# B&R Automation Studio project NAELD004C00R10L518F00 (part 47)

#### Act_InitLocal.st
```iecst
(** 2019-04-16 **)
ACTION Act_InitLocal:

	//Input Reference Link To Local Variable
	p_udiRstErr ACCESS ADR(udiRstErr);
	p_bEn ACCESS ADR(bEn);
	p_bDis ACCESS ADR(bDis);
	p_bRun ACCESS ADR(bRun);
	p_bStop ACCESS ADR(bStop);
	p_bStep ACCESS ADR(bStep);

	p_sProgNm ACCESS ADR(sProgNm);
	p_bNtSettingsLoadDone ACCESS ADR(bNtSettingsLoadDone);

	p_usiMagConv ACCESS ADR(usiMagConv);
	p_bInfoEn ACCESS ADR(bInfoEn);
	p_bInfoMag1Mty ACCESS ADR(bInfoMag1Mty);
	p_bInfoMag2Mty ACCESS ADR(bInfoMag2Mty);
	p_bInfoMag3Mty ACCESS ADR(bInfoMag3Mty);

	pa_bMagDis ACCESS ADR(a_bMagDis);

	p_bNewMag ACCESS ADR(bNewMag);
	p_bRlsMag ACCESS ADR(bRlsMag);

	p_bUSAllow ACCESS ADR(bUSAllow);
	p_tyBufferStat1 ACCESS ADR(tyBufferStat1);
	p_tyBufferStat2 ACCESS ADR(tyBufferStat2);
	p_tyBufferStat3 ACCESS ADR(tyBufferStat3);
	p_tyBufferStat4 ACCESS ADR(tyBufferStat4);

	p_bMagClampRS1 ACCESS ADR(bMagClampRS1);
	p_bMagClampRS2 ACCESS ADR(bMagClampRS2);
	p_bMagClampRS3 ACCESS ADR(bMagClampRS3);
	p_bMagClampRS4 ACCESS ADR(bMagClampRS4);

	p_bMagEntrySen1 ACCESS ADR(bMagEntrySen1);
	p_bMagEntrySen2 ACCESS ADR(bMagEntrySen2);
	p_bMagEntrySen3 ACCESS ADR(bMagEntrySen3);
	p_bMagEntrySen4 ACCESS ADR(bMagEntrySen4);

	p_bMagPresentSen1 ACCESS ADR(bMagPresentSen1);
	p_bMagPresentSen2 ACCESS ADR(bMagPresentSen2);
	p_bMagPresentSen3 ACCESS ADR(bMagPresentSen3);
	p_bMagPresentSen4 ACCESS ADR(bMagPresentSen4);

	p_bBufferMagPresent1 ACCESS ADR(bBufferMagPresent1);
	p_bBufferMagPresent2 ACCESS ADR(bBufferMagPresent2);
	p_bBufferMagPresent3 ACCESS ADR(bBufferMagPresent3);
	p_bBufferMagPresent4 ACCESS ADR(bBufferMagPresent4);

	p_dtBufferMagPresentTm1 ACCESS ADR(dtBufferMagPresentTm1);
	p_dtBufferMagPresentTm2 ACCESS ADR(dtBufferMagPresentTm2);
	p_dtBufferMagPresentTm3 ACCESS ADR(dtBufferMagPresentTm3);
	p_dtBufferMagPresentTm4 ACCESS ADR(dtBufferMagPresentTm4);

	p_eBufferStat ACCESS ADR(eBufferStat);
	p_eBufferStatus ACCESS ADR(eBufferStatus);

	p_eMagConv2ClpStat ACCESS ADR(eMagConv2ClpStat);
	p_eMagConv2ClpStatus ACCESS ADR(eMagConv2ClpStatus);
	p_bMagConv2ClpHvMag ACCESS ADR(bMagConv2ClpHvMag);

	p_eDSSMEMAStat ACCESS ADR(eDSSMEMAStat);
	p_eDSSMEMAStatus ACCESS ADR(eDSSMEMAStatus);
	p_bDSSMEMAConvStart ACCESS ADR(bDSSMEMAConvStart);

	p_eAGVMagStat ACCESS ADR(eAGVMagStat);
	p_eAGVMagStatus ACCESS ADR(eAGVMagStatus);
	p_bAGVMagMcRunRdy ACCESS ADR(bAGVMagMcRunRdy);
	p_tyAGVToDTMag ACCESS ADR(tyAGVToDTMag);

	p_eTrolleyLckStat ACCESS ADR(eTrolleyLckStat);
	p_eTrolleyLckStatus ACCESS ADR(eTrolleyLckStatus);

END_ACTION
```

#### Act_Link.st
```iecst
(** 2018-12-11 **)
ACTION Act_Link:

	IF p_eLinkMag = LDMagQuadruple = FALSE THEN
		//Sensor
		p_bMagPresentSen1	:= p_bLinkDIMagPresentSen1 OR p_bLinkMagConv2Clp1MtrIn OR p_bLinkMagConv2Clp1MtrOut;
		p_bMagPresentSen2	:= p_bLinkDIMagPresentSen2 OR p_bLinkMagConv2Clp2MtrIn OR p_bLinkMagConv2Clp2MtrOut;
		p_bMagPresentSen3	:= p_bLinkDIMagPresentSen3 OR p_bLinkMagConv2Clp3MtrIn OR p_bLinkMagConv2Clp3MtrOut;
		p_bMagPresentSen4	:= p_bLinkDIMagPresentSen4 OR p_bLinkMagConv2Clp4MtrIn OR p_bLinkMagConv2Clp4MtrOut;

		//Clamp RS
		p_bMagClampRS1 		:= (p_bLinkFixedMagClampRS1 AND p_bLinkRmtMagClampRS1) OR p_bLinkNewMagVerified1;
		p_bMagClampRS2		:= (p_bLinkFixedMagClampRS2 AND p_bLinkRmtMagClampRS2) OR bNewMagVerified;
		p_bMagClampRS3		:= (p_bLinkFixedMagClampRS3 AND p_bLinkRmtMagClampRS3) OR p_bLinkNewMagVerified3;
		p_bMagClampRS4		:= (p_bLinkFixedMagClampRS4 AND p_bLinkRmtMagClampRS4) OR p_bLinkNewMagVerified4;

	ELSE
		IF p_eLinkMag = LDMagQuadruple THEN
			CASE p_usiLinkMod OF
				0,1:
					//Sensor
					p_bMagPresentSen1	:= p_bLinkDIMagPresentSen1 OR p_bLinkMagConv2Clp1MtrIn OR p_bLinkMagConv2Clp1MtrOut;
					p_bMagPresentSen2	:= p_bLinkDIMagPresentSen2 OR p_bLinkMagConv2Clp2MtrIn OR p_bLinkMagConv2Clp2MtrOut;
					p_bMagPresentSen3	:= p_bLinkDIMagPresentSen3 OR p_bLinkMagConv2Clp3MtrIn OR p_bLinkMagConv2Clp3MtrOut;
					p_bMagPresentSen4	:= p_bLinkDIMagPresentSen4 OR p_bLinkMagConv2Clp4MtrIn OR p_bLinkMagConv2Clp4MtrOut;

					//Clamp RS
					p_bMagClampRS1 		:= (p_bLinkFixedMagClampRS1 AND p_bLinkRmtMagClampRS1) OR p_bLinkNewMagVerified1;
					p_bMagClampRS2		:= (p_bLinkFixedMagClampRS2 AND p_bLinkRmtMagClampRS2) OR bNewMagVerified;
					p_bMagClampRS3		:= (p_bLinkFixedMagClampRS3 AND p_bLinkRmtMagClampRS3) OR p_bLinkNewMagVerified3;
					p_bMagClampRS4		:= (p_bLinkFixedMagClampRS4 AND p_bLinkRmtMagClampRS4) OR p_bLinkNewMagVerified4;

				2:
					//Sensor
					p_bMagPresentSen1	:= p_bLinkDIMagPresentSen1 OR p_bLinkMagConv2Clp1MtrIn OR p_bLinkMagConv2Clp1MtrOut;
					p_bMagPresentSen2	:= p_bLinkDIMagPresentSen2 OR p_bLinkMagConv2Clp2MtrIn OR p_bLinkMagConv2Clp2MtrOut;
					p_bMagPresentSen3	:= FALSE;
					p_bMagPresentSen4	:= FALSE;

					//Clamp RS
					p_bMagClampRS1 		:= (p_bLinkFixedMagClampRS1 AND p_bLinkRmtMagClampRS1) OR p_bLinkNewMagVerified1;
					p_bMagClampRS2		:= (p_bLinkFixedMagClampRS2 AND p_bLinkRmtMagClampRS2) OR bNewMagVerified;
					p_bMagClampRS3		:= FALSE;
					p_bMagClampRS4		:= FALSE;

			END_CASE
		END_IF
	END_IF

	//Mag Exchange Mode
	CASE p_eLinkMcParamMagExMode OF
		McSetMagXcAutoManMode:
			bMagManEx := TRUE;
			bMagAutoEx := TRUE;

		McSetMagXcAutoMode:
			bMagManEx := FALSE;
			bMagAutoEx := TRUE;

		McSetMagXcManMode:
			bMagManEx := TRUE;
			bMagAutoEx := FALSE;

	END_CASE

	//New magazine auto detection at inlet sensor
	fbMagAutoDetTm(IN := p_bLinkDIMagEntrySen OR p_bLinkDIMagPresentSen2, PT := DINT_TO_TIME(p_bLinkMcParamMagAutoDetTm));
	IF fbMagAutoDetTm.Q AND bMagManEx THEN
		bNewMagAutoDetected := TRUE;
	ELSE
		bNewMagAutoDetected := FALSE;
	END_IF

	//Front or rear lane magazine mode
	IF p_eLinkMag = LDMagQuadruple THEN
		CASE p_usiLinkMod OF
			0,2:
				usiMagModel := p_bLinkMagRcpCurrRcpMagModel;

			1:
				usiMagModel := p_bLinkMagRcpCurrRcpMagModel1;
		END_CASE

	ELSE
		usiMagModel := p_bLinkMagRcpCurrRcpMagModel;

	END_IF

	IF p_bLinkNtParamMagModelAutoVerify THEN
		IF usiMagModel = 0  //CAB706.2
			AND p_bDIMagConvHeightSen = TRUE
			AND p_bDIMagConvSelUnclampRS = FALSE
			AND p_bDIMagConvCAB717Sen = FALSE
			AND p_bDIMagConvSmallSen
			THEN
			bNewMagVerified:= TRUE;

		ELSIF  usiMagModel = 1 //CAB716.2
			AND p_bDIMagConvHeightSen = FALSE
			AND p_bDIMagConvSelUnclampRS = FALSE
			AND p_bDIMagConvCAB717Sen = FALSE
			AND p_bDIMagConvSmallSen
			THEN
			bNewMagVerified:= TRUE;

		ELSIF  usiMagModel = 2 //CAB717.2
			AND p_bDIMagConvHeightSen = FALSE
			AND p_bDIMagConvSelUnclampRS
			AND p_bDIMagConvCAB717Sen
			AND p_bDIMagConvLargeSen
			THEN
			bNewMagVerified:= TRUE;
		ELSE
			bNewMagVerified:= FALSE;
		END_IF
	ELSE
		bNewMagVerified:= TRUE;
	END_IF

	bAIVInPos := p_tyAGVToDTMag.bVEHInPos2 OR p_bDISOTRcv;

	IF p_bBufferMagRemoved THEN
		bManualUnloadMag := FALSE;
	END_IF

	IF EDGEPOS(p_bOpsTravLifULUpdatePullSlot) THEN
		bOpsTravLifULUpdatePullSlot := TRUE;
	ELSIF p_bOpsTravLifULUpdatePullSlot = FALSE THEN
		bOpsTravLifULUpdatePullSlot := FALSE;
	END_IF

	//Auto recipe
	IF p_bNtParamAutoRcpPrep THEN
		p_bUSAllow := NOT(p_bMagPropDiffBlk); //false
//		p_bAdaptFollowerBlk := p_sProdRcpCurrRcp1Name <>  p_sProdRcpCrZ2RcpNm;
	ELSE
		p_bUSAllow ACCESS p_Follower1USAllow;
//		p_bAdaptFollowerBlk := FALSE;
	END_IF

	//Trolley lock feature
	IF p_bLinkTrolleyLckPrep THEN
		fbTrllySenOff(IN:= p_bTrolleyPreSen=FALSE);
		IF EDGEPOS(p_bTrolleyPreSen) THEN
			eTrolleyLck :=  PneuActExt;
			bTrllyRetDone := FALSE;
		ELSIF eGotoOpsStep = MagConvLDStepMagUSComm AND eOpsStep = MagConvLDStepMagExitedWait OR p_bUITrolleyUnlck THEN
			eTrolleyLck :=  PneuActRet;
		ELSIF NOT(p_bTrolleyPreSen) AND fbTrllySenOff.Q AND bTrllyRetDone = FALSE THEN
			eTrolleyLck :=  PneuActRet;
			bTrllyRetDone := TRUE;
		END_IF
		IF p_eTrolleyLckStat = PneuActRet OR  p_eTrolleyLckStat = PneuActExt AND p_eTrolleyLckStatus = Done THEN
			eTrolleyLck :=  PneuActIdle;
			p_bUITrolleyUnlck := FALSE; //bi-dir
		END_IF
	END_IF
END_ACTION
```

#### Init.st
```iecst
(** 2019-03-25 **)
PROGRAM _INIT

	(* Always Change If Project Change *)

	//Physical Configuration
	usiMagConv	:= 2;

	//Pass Address To Global Address For External Use
	//Action, State & Status

	//Alarm
	p_OpsMagConvLD2AlmData	:= ADR(tyAlmData);
	p_OpsMagConvLD2AlmData1	:= ADR(tyAlmData1);

	//Output
	p_OpsMagConvLD2StepTxt	:= ADR(sStepTxt);
	p_OpsMagConvLD2Paused	:= ADR(bPaused);

	p_OpsMagConvLD2BufferAct		:= ADR(eBufferAct);
	p_OpsMagConvLD2MagConv2ClpAct	:= ADR(eMagConv2ClpAct);
	p_OpsMagConvLD2DSSMEMAAct		:= ADR(eDSSMEMAAct);
	p_OpsMagConvLD2AGVMagAct		:= ADR(eAGVMagAct);
	p_OpsMagConvLD2SafetyBarAct			:= ADR(eSafetyBarAct);

	p_OpsMagConvLD2InitDone				:= ADR(bOpsInitDone);
	p_OpsMagConvLD2MagBffrAvl			:= ADR(bMagBffrAvl);
	p_OpsMagConvLD2NewMagAllw			:= ADR(bNewMagAllw);
	p_OpsMagConvLD2RlsMagAllw			:= ADR(bRlsMagAllw);
	p_OpsMagConvLD2StepMagExitedWait	:= ADR(bStepMagExitedWait);
	p_OpsMagConvLD2StepUSCom			:= ADR(bStepMagUSCom);

	p_OpsMagConvLD2StepSelClampCtrl		:= ADR(eSelClampCtrl);

	p_OpsMagConvLD2NewMagVerified		:= ADR(bNewMagVerified);
	p_OpsMagConvLD2MagMtyExit			:= ADR(bStepMagMtyExit);
	p_OpsMagConvLD2IncorrectMagModel    := ADR(bIncorrectMagazineModel);
	p_OpsMagConvLD2MagSizeL    			:= ADR(bMagSizeLarge);

	p_OpsMagConvLD2USSOTAct			:= ADR(eUSSOTAct);
	p_OpsMagConvLD2DSSOTAct			:= ADR(eDSSOTAct);

	p_OpsMagConvLD2ExitedWait			:= ADR(bMagExitedWait);
	p_OpsMagConvLD2DSCom				:= ADR(bStepDSCom);
	p_OpsMagConvLD2AGVCommRdy			:= ADR(bAGVCommRdy);

	p_OpsMagConvLD2UnclmpDone			:= ADR(bPneuUnclmpDone);
	p_OpsMagConvLD2MagAllwGo			:= ADR(udiMagAllwGo);
	p_OpsMagConvLD2QueryWO 				:= ADR(bQueryWO);
	p_OpsMagConvLD2ReadRFID				:= ADR(bReadRFID);
	p_OpsMagConvLD2WriteRFID			:= ADR(bWriteRFID);
	p_OpsMagConvLD2ExtDelAutoRcp		:= ADR(bExitDelAutoRcp);
	p_OpsMagConvLD2RlsMagUmask			:= ADR(bRlsMagBtnUnmask);
	p_OpsMagConvLD2ExtMes				:= ADR(bExtMesStdByChk);
	p_OpsMagConvLD2HModChgDone			:= ADR(bHCommModChgDone);
	p_OpsMagConvLD2TrolleyLck			:= ADR(eTrolleyLck);

	(* Always Change If Project Change *)

END_PROGRAM
```

#### Program Logical/Operations/OpsMagConvLD2/Sequence

##### Act_LogStep.st
```iecst
(** 2019-03-25 **)
ACTION Act_LogStep:

//log
	IF EDGEPOS (bClsLog) THEN
		memset(ADR(logStep),0,SIZEOF(logStep));
		logIndexStep := 0;
		bClsLog := FALSE;
	END_IF

	blog := eOpsStep <> eGotoOpsStepDummy;

	IF blog THEN
		logStep[logIndexStep] := eOpsStep;
		logIndexStep := logIndexStep + 1;
		IF logIndexStep > SIZEOF(logStep)/SIZEOF(logStep[0]) -1 THEN
			logIndexStep := 0;
		END_IF
	END_IF

	eGotoOpsStepDummy := eOpsStep;

END_ACTION
```

##### Act_OpsInfo.st
```iecst
ACTION Act_OpsInfo:

	//Reset
	udiStatus1	:= 0;

	//Magazine Verification Warning
	fbMagRemovedTm(IN:= p_bMagPresentSen = FALSE AND p_bLocalMagEntrySen = FALSE AND p_bBufferMagRemoved);
	IF fbMagRemovedTm.Q OR bNewMagVerified THEN
		bNewMagVerifyStarted := FALSE;
	END_IF

	fbVerifyWarningDelay(IN:= bNewMagVerifyStarted AND bNewMagVerified = FALSE AND bStepMagVerification = FALSE);

	IF fbVerifyWarningDelay.Q AND p_tyBufferStat2.bBffrMty = FALSE THEN
		IF bManualUnloadMag = FALSE THEN
			CASE usiMagModel OF
				0: //CAB706.2
					IF bWrongHeight THEN
						udiStatus1	:= 10005;
					ELSIF p_bDIMagConvHeightSen = FALSE THEN
						bWrongHeight := TRUE;

					ELSIF bWrongWidth THEN
						udiStatus1	:= 10004;
					ELSIF p_bDIMagConvSelUnclampRS
						OR p_bDIMagConvCAB717Sen
						OR p_bDIMagConvSmallSen = FALSE
						THEN
						bWrongWidth := TRUE;
					END_IF

				1: //CAB716.2
					IF bWrongHeight THEN
						udiStatus1	:= 10005;
					ELSIF p_bDIMagConvHeightSen = TRUE THEN
						bWrongHeight := TRUE;

					ELSIF bWrongWidth THEN
						udiStatus1	:= 10004;
					ELSIF p_bDIMagConvSelUnclampRS
						OR p_bDIMagConvCAB717Sen
						OR p_bDIMagConvSmallSen = FALSE
						THEN
						bWrongWidth := TRUE;
					END_IF

				2: //CAB717.2
					IF bWrongHeight THEN
						udiStatus1	:= 10005;
					ELSIF p_bDIMagConvHeightSen THEN
						bWrongHeight := TRUE;

					ELSIF bWrongWidth THEN
						udiStatus1	:= 10004;
					ELSIF p_bDIMagConvSelUnclampRS = FALSE
						OR p_bDIMagConvCAB717Sen = FALSE
						OR p_bDIMagConvLargeSen
						THEN
						bWrongWidth := TRUE;

					END_IF

			END_CASE
		ELSIF bManualUnloadMag THEN
			udiStatus1	:= 10006;
		END_IF

	ELSIF 	udiStatus1 <> 10004
		AND udiStatus1 <> 10005
		AND p_tyBufferStat2.bBffrMty = FALSE
		AND bStepMagExitedWait
		AND p_bLocalMagEntrySen
		THEN
		udiStatus1	:= 10006;
		bManualUnloadMag := TRUE;
	ELSE
		bWrongHeight := FALSE;
		bWrongWidth	:= FALSE;
	END_IF

	bIncorrectMagazineModel := udiStatus1 = 10004 OR udiStatus1 = 10005;

	//----------------------------Siemens MES -------------------------------------//
	IF (udiStatus1 = 0) AND p_eNtParamCustomerReq = Siemens OR p_eNtParamCustomerReq = We_Fabricate THEN
		IF eOpsStep = MagConvLDStepMagExtMESStdByChk THEN	 //we_fab no use
			IF NOT(fbWriteRFIDTO.Q) THEN
				udiStatus1 := 10014;
			ELSIF fbWriteRFIDTO.Q THEN
				udiStatus1 := 10015;
			END_IF
			IF (fbMagRemovedTm.Q ) THEN
				fbWriteRFIDTO(IN:= FALSE);
			END_IF
		ELSIF eOpsStep = MagConvLDStepMagEntMESStdByChk THEN
			IF p_tyResponseFromMES.iAcceptCondition < 0 THEN
				udiStatus1 := 10016; //wrong magazine position x.Press Release Magazine To Continue.
			END_IF
		END_IF

	END_IF

END_ACTION
```

##### Act_OpsInitial.st
```iecst
(** 2019-01-16 **)
ACTION Act_OpsInitial:

	eOpsStep		:= MagConvLDStepNA;
	eGotoOpsStep	:= MagConvLDStepInitMag;

	bOpsInitDone		:= FALSE;
	bMagBffrAvl			:= FALSE;
	bNewMagAllw			:= FALSE;
	bRlsMagAllw			:= FALSE;
	bStepMagExitedWait	:= FALSE;
	bHCommModChgDone 	:= FALSE;

END_ACTION
```

##### Act_OpsRun.st
```iecst
(** 2019-04-16 **)
ACTION Act_OpsRun:
	Act_LogStep;

	IF p_bOpsTravLifErrCmdUnclmp THEN //from travLif width chk error
		eMagConv2ClpAct :=	MagConv2ClpActStopClpr;

		IF (p_eMagConv2ClpStatus = Done AND p_eMagConv2ClpStat = MagConv2ClpActStopClpr) THEN

			eMagConv2ClpAct	:= MagConv2ClpActIdle;
			bPneuUnclmpDone := TRUE; //to travlif
		END_IF
	END_IF

	IF eGotoOpsStep <> eOpsStep THEN

		CASE eGotoOpsStep OF
			MagConvLDStepSelClampCtrl:
				IF p_bMagOrientChkSenPrep THEN
					//checking orientation of mag
					IF p_bMagHeightDetEn AND p_bMagHeightDetPrep THEN

						IF p_bMag2OrientationChkSen1 AND p_bMagHeightDetSen2 THEN // Magazine Type Check with height Detection Sensor
							eOpsStep := eGotoOpsStep;
						ELSE
							eMagConv2ClpAct :=	MagConv2ClpActStopClpr;

							IF (p_eMagConv2ClpStatus = Done AND p_eMagConv2ClpStat = MagConv2ClpActStopClpr) THEN

								eMagConv2ClpAct	:= MagConv2ClpActIdle;
								eStatus		:= Error;
								udiStatus	:= 10008;	//'Wrong Magazine Orientation Placed Or Wrong Magazine Loaded'
							END_IF
						END_IF

					ELSE

					IF p_bMag2OrientationChkSen1  AND NOT p_bMagHeightDetSen2 THEN //Without Check Height Detection Sensor
						eOpsStep := eGotoOpsStep;
					ELSE
						eMagConv2ClpAct :=	MagConv2ClpActStopClpr;
						eSelClampCtrl := PneuActExt; //unclmp
						IF (p_eMagConv2ClpStatus = Done AND p_eMagConv2ClpStat = MagConv2ClpActStopClpr) THEN

							eMagConv2ClpAct	:= MagConv2ClpActIdle;
							eStatus		:= Error;
							udiStatus	:= 10008;	//'Wrong Magazine Orientation Placed Or Wrong Magazine Loaded'
						END_IF
					END_IF
					END_IF
				ELSIF p_bLinkTrolleyLckPrep THEN
					IF p_bSlotLckSenMag THEN
						eOpsStep := eGotoOpsStep;
						fbSltLckSenFailTmr(IN:= FALSE);
					ELSIF fbSltLckSenFailTmr.Q THEN
						eMagConv2ClpAct :=	MagConv2ClpActStopClpr;

						IF (p_eMagConv2ClpStatus = Done AND p_eMagConv2ClpStat = MagConv2ClpActStopClpr) THEN
							fbSltLckSenFailTmr(IN:= FALSE);

							eMagConv2ClpAct	:= MagConv2ClpActIdle;
							eStatus		:= Error;
							udiStatus	:= 10010;	//'Magazine Transport Lock Slot Is Locked.'
						END_IF
					ELSE
						fbSltLckSenFailTmr(IN:= TRUE);
					END_IF
				ELSE
					eOpsStep	:= eGotoOpsStep;
				END_IF

			MagConvLDStepMagExitClampCtrl: //For Siemen
				IF p_eNtParamCustomerReq = Siemens AND (eOpsStep <> MagConvLDStepMagExtMESStdByChk )
					AND (p_tyLocalBufferStat.bBffrMty OR p_bDISOTAGVReady)
					AND NOT(iMagMESAcptCond < 0) AND p_bMcParamMesRFIDEn THEN
					eOpsStep := MagConvLDStepMagExtMESStdByChk;
					eGotoOpsStep := MagConvLDStepMagExtMESStdByChk; //exit mes
					//ePrevStepBeforeMESStdBy := MagConvLDStepMagExitClampCtrl;
				ELSE
					bExitDelAutoRcp := TRUE; 									//Clear the rcp and calc pitch
					eOpsStep	:= eGotoOpsStep;
				END_IF

			MagConvLDStepMagExitMnl:
				IF p_bRlsMag AND  p_eNtParamCustomerReq = Siemens AND eOpsStep <> MagConvLDStepMagExtMESStdByChk
					AND eOpsStep <> MagConvLDStepMagEntMESStdByChk AND p_bMcParamMesRFIDEn THEN
					eGotoOpsStep := MagConvLDStepMagExtMESStdByChk; //exit mes
				ELSE
					IF eOpsStep = MagConvLDStepMagExtMESStdByChk THEN
						ePrevStepBeforeMESStdBy := MagConvLDStepMagExitMnl;
					END_IF
					IF p_eNtParamCustomerReq = We_Fabricate  AND p_bMcParamMesRFIDEn THEN
						bExitDelAutoRcp := TRUE;
					END_IF
					eOpsStep	:= eGotoOpsStep;
				END_IF

			ELSE
				eOpsStep	:= eGotoOpsStep;

		END_CASE

	END_IF

	IF eOpsStep = eGotoOpsStep THEN

		IF bPaused = FALSE THEN

			CASE eOpsStep OF

				MagSetupULStepInitPneu:
					sStepTxt	:= 'Initializing Pneumatic';

					p_usiMagConv := 2;
					CASE p_usiMagConv OF
						1:
							p_tyLocalBufferStat ACCESS ADR(p_tyBufferStat1);
							p_bLocalMagEntrySen ACCESS ADR(p_bMagEntrySen1);
							p_bLocalBufferMagPresent ACCESS ADR(p_bBufferMagPresent1);
							p_dtLocalBufferMagPresentTm ACCESS ADR(p_dtBufferMagPresentTm1);
						2:
							p_tyLocalBufferStat ACCESS ADR(p_tyBufferStat2);
							p_bLocalMagEntrySen ACCESS ADR(p_bMagEntrySen2);
							p_bLocalBufferMagPresent ACCESS ADR(p_bBufferMagPresent2);
							p_dtLocalBufferMagPresentTm ACCESS ADR(p_dtBufferMagPresentTm2);
						3:
							p_tyLocalBufferStat ACCESS ADR(p_tyBufferStat3);
							p_bLocalMagEntrySen ACCESS ADR(p_bMagEntrySen3);
							p_bLocalBufferMagPresent ACCESS ADR(p_bBufferMagPresent3);
							p_dtLocalBufferMagPresentTm ACCESS ADR(p_dtBufferMagPresentTm3);
						4:
							p_tyLocalBufferStat ACCESS ADR(p_tyBufferStat4);
							p_bLocalMagEntrySen ACCESS ADR(p_bMagEntrySen4);
							p_bLocalBufferMagPresent ACCESS ADR(p_bBufferMagPresent4);
							p_dtLocalBufferMagPresentTm ACCESS ADR(p_dtBufferMagPresentTm4);
					END_CASE
					IF p_bProjLifTravMnlLoad = FALSE THEN
						eSafetyBarAct	:= PneuActExt;
					ELSE
						eGotoOpsStep := MagConvLDStepMagUSComm;
					END_IF
					IF (p_eSafetyBarStatus = Done AND p_eSafetyBarStat = PneuActExt) THEN
						eSafetyBarAct	:= PneuActIdle;
						eGotoOpsStep	:= MagConvLDStepInitMag;

						bPaused	:= p_bStop OR p_bStep;
					END_IF

				MagConvLDStepInitMag:
					sStepTxt	:= 'Initializing Magazine';
					IF p_bProjLifTravMnlLoad = TRUE THEN
						eGotoOpsStep := MagConvLDStepMagUSComm;
					ELSIF bMagExitedWait THEN
						eGotoOpsStep	:= MagConvLDStepMagExitedWait;
						//eGotoOpsStep	:= MagConvLDStepInitMagEnt;
					ELSIF (ePrevStepBeforeMESStdBy = MagConvLDStepMagExitMnl AND p_bLinkDIMagPresentSen2) OR (p_bHCommModChg AND p_bLinkDIMagPresentSen2)THEN
						eGotoOpsStep	:= MagConvLDStepMagExitMnl;
					ELSIF p_bNtParamAutoRcpPrep AND p_bHermesSvyPrep AND p_bMcParamHermesSvyEn THEN
						bHCommModChgDone := TRUE; //to UI
						eGotoOpsStep	:= MagConvLDStepInitMagConv;
					ELSE
						bHCommModChgDone := TRUE; //to UI
						eGotoOpsStep	:= MagConvLDStepInitSetMagFull;
					END_IF

					bPaused	:= p_bStop OR p_bStep;

				MagConvLDStepInitMagEnt:
					sStepTxt	:= 'Initializing Magazine Conveyor';
					eMagConv2ClpAct	:= MagConv2ClpActInit;
					IF (p_eMagConv2ClpStatus = Done AND p_eMagConv2ClpStat = MagConv2ClpActInit) THEN
						eMagConv2ClpAct	:= MagConv2ClpActIdle;
						IF p_bMagConv2ClpHvMag = FALSE THEN
							eGotoOpsStep	:= MagConvLDStepMagUSComm;
						ELSE
							eGotoOpsStep	:= MagConvLDStepInitMagFixClp;
						END_IF
					END_IF

				MagConvLDStepInitMagFixClp:
					sStepTxt	:= 'Initializing Fixed Clamp';
					eMagConv2ClpAct	:= MagConv2ClpActFixClprClamp;
					IF (p_eMagConv2ClpStatus = Done AND p_eMagConv2ClpStat = MagConv2ClpActFixClprClamp) THEN
						eMagConv2ClpAct	:= MagConv2ClpActIdle;
						IF bMagAutoEx THEN
							eDSSOTAct	:= SOTActRun;
						ELSE
							eDSSOTAct	:= SOTActIdle;
						END_IF

						IF p_bDIMagConvCAB717Sen THEN
							bMagSizeLarge := TRUE;
						ELSE
							bMagSizeLarge := FALSE;
						END_IF
						eGotoOpsStep	:= MagConvLDStepSelClampCtrl;
					END_IF

				MagConvLDStepInitSetMagFull	:
					sStepTxt	:= 'Set Magazine Full';
					IF bSetMagFull AND p_tyBufferStat2.diTtlBrdCap = 1 THEN
						eBufferAct := BufferActSetFull;
						IF p_eBufferStat = BufferActSetFull AND p_eBufferStatus = Done THEN
							bSetMagFull := FALSE;
							eBufferAct := BufferActIdle;
							eGotoOpsStep	:= MagConvLDStepInitMagConv;
						END_IF
					ELSIF bSetMagFull AND p_tyBufferStat2.diTtlBrdCap <> 1 THEN
						bSetMagFull := FALSE;
						eBufferAct := BufferActIdle;
						eGotoOpsStep	:= MagConvLDStepInitMagConv;
					ELSE
						bSetMagFull := FALSE;
						eBufferAct := BufferActIdle;
						eGotoOpsStep	:= MagConvLDStepInitMagConv;
					END_IF
					bPaused	:= p_bStop OR p_bStep;

				MagConvLDStepInitMagConv:
					sStepTxt	:= 'Initializing Magazine Conveyor';

					eMagConv2ClpAct	:= MagConv2ClpActInitStopClp;
					eSelClampCtrl := PneuActExt;

					IF (p_eMagConv2ClpStatus = Done AND p_eMagConv2ClpStat = MagConv2ClpActInitStopClp)
						AND (p_eSelClampCtrlStat = PneuActExt AND p_eSelClampCtrlStatus = Done)
						THEN
						eSelClampCtrl	:= PneuActIdle;
						eMagConv2ClpAct	:= MagConv2ClpActIdle;

						IF p_bMagConv2ClpHvMag = FALSE THEN
							eGotoOpsStep	:= MagConvLDStepMagUSComm;
							bExitDelAutoRcp := TRUE;
							usiAccWO := 0;
							ePrevStepBeforeMESStdBy := MagConvLDStepNA; //finish exit from extMes
						ELSE
						//	eGotoOpsStep		:= MagConvLDStepBffrStatChk;
							eGotoOpsStep		:= MagConvLDStepSelClampCtrl;
						END_IF

						bPaused	:= p_bStop OR p_bStep;

					END_IF

				MagConvLDStepSafetyBarExtCtrl:
					eSafetyBarAct	:= PneuActExt;

					IF(p_eSafetyBarStatus = Done AND p_eSafetyBarStat = PneuActExt)
						THEN
						eSafetyBarAct	:= PneuActIdle;
						eGotoOpsStep	:= MagConvLDStepMagUSComm;
					END_IF

				MagConvLDStepMagUSComm:
					sStepTxt	:= 'Communicating AIV And Ready Transport In Magazine';

					eAGVMagAct	:= AGVMagActEnter;
					IF bMagAutoEx THEN
						eUSSOTAct	:= SOTActRun;
					ELSE
						eUSSOTAct	:= SOTActIdle;
					END_IF
					eDSSOTAct	:= SOTActIdle;
					bMagSizeLarge := FALSE;
					bMagExitedWait	:= FALSE;

					IF p_bSafetyBarExtended = FALSE THEN
						eGotoOpsStep	:= MagConvLDStepSafetyBarExtCtrl;
					ELSIF p_bAGVMagMcRunRdy = TRUE OR p_bUSSOTTransporting= TRUE THEN
						eGotoOpsStep	:= MagConvLDStepMagEnt;

					ELSIF p_bNewMag = TRUE OR bNewMagAutoDetected = TRUE THEN
						eAGVMagAct		:= AGVMagActIdle;
						eGotoOpsStep	:= MagConvLDStepMagEntMnl;

					ELSE
						bPaused	:= p_bStop;

						IF bPaused = TRUE THEN
							eAGVMagAct	:= AGVMagActIdle;
							eUSSOTAct	:= SOTActIdle;
						END_IF

					END_IF

				MagConvLDStepMagEnt:

					IF p_bUSSOTConvStart THEN
						sStepTxt	:= 'Conveyor Entering Magazine To End';
						eMagConv2ClpAct	:= MagConv2ClpActEntStopClp;

					ELSIF bNewMagAutoDetected = TRUE THEN
						eAGVMagAct			:= AGVMagActIdle;
						eGotoOpsStep		:= MagConvLDStepMagEntMnl;

					ELSIF p_bUSSOTConvStop THEN
						sStepTxt	:= 'Conveyor Stopping';
						eMagConv2ClpAct	:= MagConv2ClpActStopClpr;
						IF (p_eMagConv2ClpStatus = Done AND p_eMagConv2ClpStat = MagConv2ClpActEntStopClp) THEN
							eMagConv2ClpAct		:= MagConv2ClpActIdle;

						END_IF
					END_IF

					IF (p_eMagConv2ClpStatus = Done AND p_eMagConv2ClpStat = MagConv2ClpActEntStopClp) THEN
						eAGVMagAct			:= AGVMagActIdle;
						eMagConv2ClpAct		:= MagConv2ClpActIdle;
						eUSSOTAct			:= SOTActIdle;
						eGotoOpsStep		:= MagConvLDStepSelClampCtrl;
						bPaused	:= p_bStop OR p_bStep;

					ELSE

					END_IF

				MagConvLDStepMagEntMnl:
					sStepTxt	:= 'Magazine Conveyor Entering Magazine Manually';
					IF p_bProjLifTravMnlLoad = FALSE THEN
						eMagConv2ClpAct	:= MagConv2ClpActEntStopClp ;
					ELSE
						eGotoOpsStep		:= MagConvLDStepSelClampCtrl;
					END_IF
					IF p_eMagConv2ClpStatus = Done AND p_eMagConv2ClpStat = MagConv2ClpActEntStopClp THEN

						eMagConv2ClpAct		:= MagConv2ClpActIdle;
						eGotoOpsStep		:= MagConvLDStepSelClampCtrl;
						eUSSOTAct			:= SOTActIdle;
						eAGVMagAct			:= AGVMagActIdle;
						bPaused	:= p_bStop OR p_bStep;
					END_IF

				MagConvLDStepSelClampCtrl:
					sStepTxt	:= 'Magazine Selection Control';
					bNewMagVerifyStarted := TRUE;
					bExitDelAutoRcp := FALSE;

					CASE p_bLinkMagRcpCurrRcpMagModel OF
						0: //CAB706.2
							IF p_bDIMagConvCAB717Sen = FALSE THEN
								eSelClampCtrl := PneuActRet;
							END_IF
							eGotoOpsStep	:= MagConvLDStepVerifyMag;

						1: //CAB716.2
							IF p_bDIMagConvCAB717Sen = FALSE THEN
								eSelClampCtrl := PneuActRet;
							END_IF
							eGotoOpsStep	:= MagConvLDStepVerifyMag;

						2: //CAB717.2
							eSelClampCtrl 	:= PneuActExt;
							eGotoOpsStep	:= MagConvLDStepVerifyMag;

					END_CASE

					bPaused	:= p_bStop OR p_bStep;

				MagConvLDStepVerifyMag:
					sStepTxt	:= 'Magazine Model Verification';

					bNewMagVerifyStarted := TRUE;
					fbWrongMagTm(IN:= bNewMagVerified = FALSE);
					IF fbWrongMagTm.Q AND NOT bMagExitedWait  THEN
						fbWrongMagTm(IN:= FALSE);
						eGotoOpsStep		:= MagConvLDStepMagExitMnl;
					ELSIF bMagExitedWait OR ePrevStepBeforeMESStdBy = MagConvLDStepMagExitMnl THEN //added extMes true
						eGotoOpsStep		:= MagConvLDStepMagExitMnl;
					ELSIF bNewMagVerified AND NOT bMagExitedWait THEN
						fbSelClmpTm(IN:= TRUE);
						IF fbSelClmpTm.Q THEN
							fbSelClmpTm(IN:= FALSE);
							eSelClampCtrl	:= PneuActIdle;
							IF (p_eNtParamCustomerReq = Siemens AND p_bMcParamHermesSvyEn AND p_bHermesSvyPrep) OR
								(p_eNtParamCustomerReq = We_Fabricate AND p_bMcParamMesRFIDEn) THEN
								IF  (iMagMESAcptCond > 0 OR usiAccWO > 0 OR bWriteRFID) AND iMagMESAcptCond <> 255 THEN
									p_bAutoRcpbMag2RcpLoaded := FALSE; //bi-dir
									eGotoOpsStep		:= MagConvLDStepBffrStatChk;
								ELSIF iMagMESAcptCond = 0  OR usiAccWO = 0 THEN
									bQueryWO := TRUE;
									eGotoOpsStep		:= MagConvLDStepMagEntMESStdByChk;
								END_IF
							ELSE
								eGotoOpsStep		:= MagConvLDStepBffrStatChk;
							END_IF
						END_IF

					END_IF

					IF p_bDIMagConvCAB717Sen THEN
						bMagSizeLarge := TRUE;
					ELSE
						bMagSizeLarge := FALSE;
					END_IF

//					IF bNewMagVerified AND p_eSelClampCtrlStatus = Done THEN
//
//						eSelClampCtrl	:= PneuActIdle;
//						eGotoOpsStep	:= MagConvLDStepBffrStatChk;
//					END_IF
					bPaused	:= p_bStop OR p_bStep;

				MagConvLDStepMagEntMESStdByChk:
					sStepTxt	:= 'Read RFID and Query Work Order';
					bReadRFID := TRUE;
					fbReadRFIDTO(IN:= bReadRFID);
					iMagMESAcptCond := INT_TO_USINT(p_tyResponseFromMES.iAcceptCondition);
					IF (p_tyResponseFromMES.iAcceptCondition > 0 AND p_eNtParamCustomerReq = We_Fabricate) OR p_bAutoRcpbMag2RcpLoaded THEN //Accept or rcv sendWO
						usiAccWO := 1;
						bQueryWO := FALSE;
						p_bAutoRcpbMag2RcpLoaded := FALSE; //bi-dir
						eGotoOpsStep := MagConvLDStepAutoRcpSetMagFull;
					//	eGotoOpsStep := MagConvLDStepBffrStatChk;
					ELSIF p_tyResponseFromMES.iAcceptCondition < 0  THEN						//No Accept (-1)
						eAGVMagAct	:= AGVMagActExit;
						IF p_bRlsMag THEN
							p_bRlsMag := FALSE; //bi-dir
							bQueryWO := FALSE;
							eGotoOpsStep	:= MagConvLDStepMagExitMnl;
						ELSIF p_bAGVMagMcRunRdy = TRUE THEN
							bQueryWO := FALSE;
							eGotoOpsStep	:= MagConvLDStepMagMtyExit;
						END_IF
					ELSIF fbReadRFIDTO.Q THEN
						sStepTxt	:= 'Wait For Read RFID';
						IF p_bRlsMag THEN
							p_bRlsMag := FALSE; //bi-dir
							bQueryWO := FALSE;
							eGotoOpsStep	:= MagConvLDStepMagExitMnl;
						END_IF
					END_IF
					IF eGotoOpsStep <> MagConvLDStepMagEntMESStdByChk THEN
						bReadRFID := FALSE;
						fbReadRFIDTO(IN:= bReadRFID);//false
					END_IF
					IF p_eNtParamCustomerReq = We_Fabricate THEN
						sStepTxt	:= 'Wait For MES feedback';
					END_IF
					bPaused	:= p_bStop OR p_bStep;

				MagConvLDStepAutoRcpSetMagFull:
					sStepTxt	:= 'Set Magazine Full';
					eBufferAct := BufferActSetFull;
					IF p_eBufferStat = BufferActSetFull AND p_eBufferStatus = Done THEN
						eBufferAct := BufferActIdle;
						IF p_ausiSvyMagAccOrder[2] = 10 OR p_ausiLCSLFMagAccOrder[2] = 10 THEN //working number
							eGotoOpsStep := MagConvLDStepBffrStatChk;
						END_IF
					END_IF
					bPaused	:= p_bStop OR p_bStep;

				MagConvLDStepBffrStatChk:
					sStepTxt	:= 'Checking Buffer Status';

					IF p_eBufferStatus = Idle THEN

						IF (p_tyLocalBufferStat.bBffrMty = TRUE OR p_bUSAllow = FALSE) THEN
							//eGotoOpsStep	:= MagConvLDStepMagMtyDSComm;
							eGotoOpsStep	:= MagConvLDStepMagExitClampCtrl;
						ELSE
							eGotoOpsStep	:= MagConvLDStepSafetyBarRetCtrl;
						END_IF

						bPaused	:= p_bStop OR p_bStep;

					END_IF

				MagConvLDStepSafetyBarRetCtrl:
					eSafetyBarAct	:= PneuActRet;

					IF (p_eSafetyBarStatus = Done AND p_eSafetyBarStat = PneuActRet) THEN
						eSafetyBarAct	:= PneuActIdle;
						eGotoOpsStep	:= MagConvLDStepPreNxtUnlBffr;

						bPaused	:= p_bStop OR p_bStep;
					END_IF

				MagConvLDStepPreNxtUnlBffr:
					sStepTxt	:= 'Computing Next Unload Buffer';

					eBufferAct	:= BufferActNxtUnload;

					IF p_eBufferStatus = Done AND p_eBufferStat = BufferActNxtUnload THEN
						eBufferAct		:= BufferActIdle;
						eGotoOpsStep	:= MagConvLDStepMagCmp;

						bPaused	:= p_bStop OR p_bStep;
					END_IF

				MagConvLDStepMagCmp:
					sStepTxt	:= 'Comparing Magazine';

					a_tyMagAllwBffrStat[1]	:= p_tyBufferStat1;
					a_tyMagAllwBffrStat[2]	:= p_tyBufferStat2;
					a_tyMagAllwBffrStat[3]	:= p_tyBufferStat3;
					a_tyMagAllwBffrStat[4]	:= p_tyBufferStat4;

					a_bMagAllwMagClamped[1]	:= p_bMagClampRS1;
					a_bMagAllwMagClamped[2]	:= p_bMagClampRS2;
					a_bMagAllwMagClamped[3]	:= p_bMagClampRS3;
					a_bMagAllwMagClamped[4]	:= p_bMagClampRS4;

					a_bMagAllwMagPresent[1]	:= p_bBufferMagPresent1 AND NOT p_bLD1ExitedWait;
					a_bMagAllwMagPresent[2]	:= p_bBufferMagPresent2 AND NOT bMagExitedWait;
					a_bMagAllwMagPresent[3]	:= p_bBufferMagPresent3 AND NOT p_bLD3ExitedWait;
					a_bMagAllwMagPresent[4]	:= p_bBufferMagPresent4 AND NOT p_bLD4ExitedWait;

					a_udiMagAllwMagPresentTm[1]	:= DT_TO_UDINT(p_dtBufferMagPresentTm1);
					a_udiMagAllwMagPresentTm[2]	:= DT_TO_UDINT(p_dtBufferMagPresentTm2);
					a_udiMagAllwMagPresentTm[3]	:= DT_TO_UDINT(p_dtBufferMagPresentTm3);
					a_udiMagAllwMagPresentTm[4]	:= DT_TO_UDINT(p_dtBufferMagPresentTm4);
					//Sorting Priority
					memset(ADR(a_udiMagAllwPriority), 0, SIZEOF(a_udiMagAllwPriority));

					IF (p_bMcParamHermesSvyEn AND p_bNtParamAutoRcpPrep) OR (p_bMcParamMesRFIDEn AND p_eNtParamCustomerReq = We_Fabricate) THEN
						FOR udi :=1 TO 3 DO
							IF p_ausiSvyMagAccOrder[udi] = 10 OR p_ausiLCSLFMagAccOrder[udi] = 10 THEN
								a_udiMagAllwPriority[udi] :=  1;
							ELSE
								a_udiMagAllwPriority[udi] := 3;
							END_IF
						END_FOR

					ELSE // standard
						FOR udi := 1 TO 4 DO
							udiCount	:= 4;
							udiCmpTm	:= a_udiMagAllwMagPresentTm[udi];

							FOR udi1 := 1 TO 4 DO
								IF a_udiMagAllwMagPresentTm[udi1] > udiCmpTm THEN
									udiCount	:= udiCount - 1;
								END_IF
							END_FOR

							a_udiMagAllwPriority[udi]	:= udiCount;
						END_FOR
						FOR udi := 4 TO 1 BY -1 DO
							FOR udi1 := 4 TO 1 BY -1 DO
								IF (udi <> udi1) AND (a_udiMagAllwPriority[udi] = a_udiMagAllwPriority[udi1]) THEN
									a_udiMagAllwPriority[udi1]	:= a_udiMagAllwPriority[udi1] - 1;
								END_IF
							END_FOR
						END_FOR
					END_IF

					//Checking Buffer Status
					memset(ADR(a_udiMagAllwSum), 0, SIZEOF(a_udiMagAllwSum));

					FOR udi := 1 TO 4 DO
						//Priority
						a_udiMagAllwSum[udi]	:= a_udiMagAllwSum[udi] + a_udiMagAllwPriority[udi];
						//Enable
						IF pa_bMagDis[udi] = FALSE THEN
							a_udiMagAllwSum[udi]	:= a_udiMagAllwSum[udi] + 1000;
						END_IF
						//Magazine Clamped
						IF a_bMagAllwMagClamped[udi] = TRUE THEN
							a_udiMagAllwSum[udi]	:= a_udiMagAllwSum[udi] + 1000;
						END_IF
						//Magazine Present
						IF a_bMagAllwMagPresent[udi] = TRUE THEN
							a_udiMagAllwSum[udi]	:= a_udiMagAllwSum[udi] + 1000;
						END_IF
						//Magazine Full
						IF a_tyMagAllwBffrStat[udi].bBffrFull = TRUE THEN
							a_udiMagAllwSum[udi]	:= a_udiMagAllwSum[udi] + 2500;
						END_IF
						//Magazine Available
						IF a_tyMagAllwBffrStat[udi].bBffrFull = FALSE AND a_tyMagAllwBffrStat[udi].bBffrMty = FALSE THEN
							a_udiMagAllwSum[udi]	:= a_udiMagAllwSum[udi] + 3000;
						END_IF
					END_FOR

					udiMagAllwGo	:= 99;

					FOR udi := 1 TO 4 DO
						//Enable + Magazine Clamped + Magazine Present + Magazine Available
						IF a_udiMagAllwSum[udi] >= 6000 THEN

							IF udiMagAllwGo <> 99 THEN
								//Priority
								IF a_udiMagAllwSum[udi] < a_udiMagAllwSum[udiMagAllwGo] THEN
									udiMagAllwGo	:= udi;
								END_IF
							ELSE
								udiMagAllwGo	:= udi;
							END_IF

						END_IF

					END_FOR

					IF udiMagAllwGo = 99 THEN

						FOR udi := 1 TO 4 DO
							//Enable + Magazine Clamped + Magazine Present + Magazine Full
							IF a_udiMagAllwSum[udi] >= 5500 THEN

								IF udiMagAllwGo <> 99 THEN
									//Priority
									IF a_udiMagAllwSum[udi] < a_udiMagAllwSum[udiMagAllwGo] THEN
										udiMagAllwGo	:= udi;
									END_IF
								ELSE
									udiMagAllwGo	:= udi;
								END_IF

							END_IF

						END_FOR

					END_IF

					IF p_bRlsMag = TRUE THEN
						eGotoOpsStep	:= MagConvLDStepMagExitMnl;

					ELSIF p_bDISOTAGVReady AND p_eNtParamCustomerReq = Siemens THEN
						eGotoOpsStep	:= MagConvLDStepMagExitClampCtrl;

					ELSIF (p_tyLocalBufferStat.bBffrMty = TRUE OR p_bUSAllow = FALSE) AND p_bInShutterExtended THEN
					//	eGotoOpsStep    := MagConvLDStepMagMtyDSComm;
						eGotoOpsStep    := MagConvLDStepMagExitClampCtrl;
					ELSE

						IF udiMagAllwGo <> 99 THEN

							IF udiMagAllwGo = p_usiMagConv (*AND p_eOpsTravLifLDPosGo = TravLifLDPosUS2*) THEN
								bMagBffrAvl		:= TRUE;
								eGotoOpsStep	:= MagConvLDStepNxtUnloadBffr;

								bPaused	:= p_bStop OR p_bStep;
							ELSE
								bPaused	:= p_bStop;
							END_IF

						ELSE
							bPaused	:= p_bStop;
						END_IF

					END_IF

				MagConvLDStepNxtUnloadBffr:
					sStepTxt	:= 'Computing Next Unload Buffer';

					eBufferAct	:= BufferActNxtUnload;

					IF p_eBufferStatus = Done AND p_eBufferStat = BufferActNxtUnload THEN
						eBufferAct		:= BufferActIdle;
						eGotoOpsStep	:= MagConvLDStepBffrDSComm;

						bPaused	:= p_bStop OR p_bStep;
					END_IF

				MagConvLDStepBffrDSComm:
					sStepTxt	:= 'Communicating Buffer Downstream';

//					IF (p_tyBufferStat2.bBffrFull OR p_bBufferMagPresent2 = FALSE)
//						AND (p_tyBufferStat3.bBffrFull OR p_bBufferMagPresent3 = FALSE)
//						THEN
//						eDSSMEMAAct	:= SMEMAActRun;
//					END_IF

					eDSSMEMAAct	:= SMEMAActRun;

					IF p_bDSSMEMAConvStart = TRUE THEN
						eGotoOpsStep	:= MagConvLDStepBffrExitBrd;

					ELSIF bOpsTravLifULUpdatePullSlot AND p_eOpsTravLifLDPosGo = TravLifLDPosUS2 THEN
						bMagBffrAvl		:= FALSE;
						IF p_tyLocalBufferStat.bBffrMty = FALSE AND p_bUIP800Press2 = FALSE THEN
							eGotoOpsStep	:= MagConvLDStepUnloadBffr;
						ELSE
							eGotoOpsStep	:= MagConvLDStepBffrStatChk;
							bMagBffrAvl		:= FALSE;
						END_IF

					ELSIF p_bRlsMag = TRUE THEN
						bMagBffrAvl		:= FALSE;
						eDSSMEMAAct		:= SMEMAActIdle;
						eGotoOpsStep	:= MagConvLDStepMagExitMnl;

					ELSIF (p_tyLocalBufferStat.bBffrMty = TRUE OR p_bUSAllow = FALSE) AND p_bInShutterExtended THEN
						bMagBffrAvl		:= FALSE;
						eDSSMEMAAct		:= SMEMAActIdle;
					//	eGotoOpsStep    := MagConvLDStepMagMtyDSComm;
						eGotoOpsStep    := MagConvLDStepMagExitClampCtrl;
					ELSE

						IF pa_bMagDis[usiMagConv] = TRUE THEN		//Checking Magazine Enable
							bMagBffrAvl		:= FALSE;
					//		eGotoOpsStep	:= MagConvLDStepMagCmp;
							eGotoOpsStep	:= MagConvLDStepPreNxtUnlBffr;

							bPaused	:= p_bStop OR p_bStep;
						ELSE
							bPaused	:= p_bStop;
						END_IF

						IF bPaused = TRUE OR pa_bMagDis[usiMagConv] = TRUE THEN
							eDSSMEMAAct	:= SMEMAActIdle;
						END_IF

					END_IF

				MagConvLDStepBffrExitBrd:
					IF p_bDSSMEMAConvStart = TRUE THEN
						sStepTxt	:= 'Transferring Board Out From Magazine';
						IF p_bRlsMag = TRUE THEN
							bMagBffrAvl		:= FALSE;
							eDSSMEMAAct		:= SMEMAActIdle;
							eGotoOpsStep	:= MagConvLDStepMagExitMnl;
						END_IF
					END_IF

					IF p_eDSSMEMAStatus = Done AND p_eDSSMEMAStat = SMEMAActRun THEN
						eDSSMEMAAct		:= SMEMAActIdle;
						//	eGotoOpsStep	:= MagConvLDStepUnloadBffr;
						IF p_tyLocalBufferStat.bBffrMty = FALSE THEN
							eGotoOpsStep	:= MagConvLDStepUnloadBffr;
						ELSE
							eGotoOpsStep	:= MagConvLDStepBffrStatChk;
							bMagBffrAvl		:= FALSE;
						END_IF
					END_IF

				MagConvLDStepUnloadBffr:
					sStepTxt	:= 'Unloading Buffer';

						eBufferAct	:= BufferActUnload;
						bOpsTravLifULUpdatePullSlot := FALSE;
						bMagBffrAvl		:= FALSE;
					IF p_eBufferStatus = Done AND p_eBufferStat = BufferActUnload THEN
						eBufferAct		:= BufferActIdle;
						bMagBffrAvl		:= FALSE;

							eGotoOpsStep	:= MagConvLDStepBffrStatChk;

						bPaused	:= p_bStop OR p_bStep;
					END_IF

				MagConvLDStepMagExtMESStdByChk:
					sStepTxt	:= 'Mag StdBy for MES response Before Exiting';
					bWriteRFID := TRUE;
					fbWriteRFIDTO(IN:= bWriteRFID ,PT:= DINT_TO_TIME(p_diRFIDTO));
					bExitDelAutoRcp := TRUE; 								//Clear the rcp and calc pitch
					IF p_tyResponseFromMES.bRFIDWriteComplete  THEN 		//Accept
//						IF ePrevStepBeforeMESStdBy = MagConvULStepMagExitMnl THEN
							eGotoOpsStep := MagConvLDStepMagExitMnl;//MagConvLDStepMagExitClampCtrl;
//						ELSIF ePrevStepBeforeMESStdBy = MagConvULStepMagExitClampCtrl THEN
//							eGotoOpsStep := MagConvLDStepMagExitClampCtrl;
//						END_IF
					ELSIF fbWriteRFIDTO.Q  THEN
						sStepTxt	:= 'MES response to Write RFID Timeout, Press Rls Mag to Manual Exit ';
						IF p_bEjectMag THEN
							eGotoOpsStep := MagConvLDStepMagExitMnl;
						END_IF
					END_IF
					IF eGotoOpsStep <> MagConvLDStepMagExtMESStdByChk THEN
						bWriteRFID := FALSE;
						fbWriteRFIDTO(IN:= bWriteRFID);

					END_IF
					bPaused	:= p_bStop OR p_bStep;

				MagConvLDStepMagExitClampCtrl:
					sStepTxt	:= 'Extending Selection Clamp';
					eSelClampCtrl := PneuActExt;
					eSafetyBarAct	:= PneuActExt;

					IF (p_eSelClampCtrlStat = PneuActExt AND p_eSelClampCtrlStatus = Done)
						AND(p_eSafetyBarStatus = Done AND p_eSafetyBarStat = PneuActExt)
						THEN
							eSelClampCtrl	:= PneuActIdle;
							eSafetyBarAct	:= PneuActIdle;
							eGotoOpsStep    := MagConvLDStepMagMtyDSComm;
							bPaused	:= p_bStop OR p_bStep;
					END_IF

				MagConvLDStepMagMtyDSComm:
					sStepTxt	:= 'Communicating AGV Machine And Ready Exit';

					eAGVMagAct	:= AGVMagActExit;
					IF bMagAutoEx THEN
						eDSSOTAct	:= SOTActRun;
					ELSE
						eDSSOTAct	:= SOTActIdle;
					END_IF

					IF p_bAGVMagMcRunRdy = TRUE THEN
						eGotoOpsStep	:= MagConvLDStepMagMtyExit;

					ELSIF p_bRlsMag = TRUE OR ((p_tyLocalBufferStat.bBffrMty OR p_bUSAllow = FALSE) AND p_bInShutterExtended) THEN
						eAGVMagAct		:= AGVMagActIdle;
						eGotoOpsStep	:= MagConvLDStepMagExitMnl;

					ELSE
						bPaused	:= p_bStop;

						IF bPaused = TRUE THEN
							eAGVMagAct	:= AGVMagActIdle;
							eDSSOTAct	:= SOTActIdle;
						END_IF

					END_IF

				MagConvLDStepMagMtyExit:
					sStepTxt	:= 'Magazine Conveyor Exiting Magazine';

					eMagConv2ClpAct	:= MagConv2ClpActExitClpr;
					eSelClampCtrl	:= PneuActExt;

					IF ((p_eAGVMagStatus = Done AND p_eAGVMagStat = AGVMagActExit)
						OR (p_eDSSOTStatus = Done AND p_eDSSOTStat = SOTActRun))
						AND (p_eMagConv2ClpStatus = Done AND p_eMagConv2ClpStat = MagConv2ClpActExitClpr)
						AND (p_eSelClampCtrlStatus = Done AND p_eSelClampCtrlStat = PneuActExt)
						THEN

						eDSSOTAct	:= SOTActIdle;
						eAGVMagAct		:= AGVMagActIdle;
						eMagConv2ClpAct	:= MagConv2ClpActIdle;
						eSelClampCtrl	:= PneuActIdle;
						eGotoOpsStep	:= MagConvLDStepMagExitedAGVWait;
						bMagSizeLarge	:= FALSE;

						bPaused	:= p_bStop OR p_bStep;
					END_IF

				MagConvLDStepMagExitedAGVWait:
					sStepTxt	:= 'Magazine Exited and Wait for AGV Leave';

					IF bAIVInPos = FALSE OR p_bBufferMagRemoved THEN
						usiAccWO := 0;
						bExitDelAutoRcp := FALSE;
						eGotoOpsStep	:= MagConvLDStepMagUSComm;
						eDSSOTAct	:= SOTActIdle;
					END_IF

					bPaused	:= p_bStop OR p_bStep;

				MagConvLDStepMagExitMnl:
					sStepTxt	:= 'Magazine Conveyor Exiting Magazine Manually';
					IF p_bProjLifTravMnlLoad = FALSE THEN
						eMagConv2ClpAct	:= MagConv2ClpActPreExitClpr;
						eSelClampCtrl	:= PneuActExt;
						eSafetyBarAct	:= PneuActExt;
					ELSE
						eGotoOpsStep    := MagConvLDStepMagExitedWait;
					END_IF
					IF ((p_eMagConv2ClpStatus = Done OR EDGENEG(p_bFixedSideDetect)) AND p_eMagConv2ClpStat = MagConv2ClpActPreExitClpr)
						AND (p_eSelClampCtrlStatus = Done AND p_eSelClampCtrlStat = PneuActExt)
						AND (p_eSafetyBarStatus = Done AND p_eSafetyBarStat = PneuActExt)
						THEN
						eSelClampCtrl	:= PneuActIdle;
						eSafetyBarAct	:= PneuActIdle;
						eMagConv2ClpAct	:= MagConv2ClpActIdle;

						eGotoOpsStep	:= MagConvLDStepMagExitedWait;

						bPaused	:= p_bStop OR p_bStep;
					END_IF

				MagConvLDStepMagExitedWait:
					sStepTxt	:= 'Magazine Exited And Waiting For Remove';
					eAGVMagAct	:= AGVMagActExit;
					IF bMagAutoEx THEN
						eDSSOTAct	:= SOTActRun;
					ELSE
						eDSSOTAct	:= SOTActIdle;
					END_IF
					bMagExitedWait	:= TRUE;
					bHCommModChgDone := TRUE; //to UI
					fbEntSenOff(IN:= p_bLocalMagEntrySen = FALSE);
					ePrevStepBeforeMESStdBy := MagConvLDStepNA; //finish exit from extMes
					iMagMESAcptCond := 0 ; //reset if 255 (-1)

					IF fbMagRemovedTm.Q OR fbEntSenOff.Q THEN
						usiAccWO := 0;
						bExitDelAutoRcp := FALSE;
						bMagExitedWait	:= FALSE;
						eGotoOpsStep	:= MagConvLDStepMagUSComm;
						eDSSOTAct	:= SOTActIdle;

					ELSIF p_bNewMag = TRUE THEN
						bMagExitedWait	:= FALSE;
						eAGVMagAct	:= AGVMagActIdle;
						eGotoOpsStep	:= MagConvLDStepMagEntMnl;
						eDSSOTAct	:= SOTActIdle;
					END_IF

					IF p_bAGVMagMcRunRdy = TRUE THEN
						eGotoOpsStep	:= MagConvLDStepMagMtyExit;
					ELSIF p_bDSSOTConvStart = TRUE THEN
						eGotoOpsStep	:= MagConvLDStepMagMtyExit;
					END_IF

					bPaused	:= p_bStop OR p_bStep;

			END_CASE

		END_IF

	END_IF

	bNewMagAllw	:= eOpsStep = MagConvLDStepMagUSComm;
	bRlsMagAllw	:= (eOpsStep = MagConvLDStepMagCmp
					OR eOpsStep = MagConvLDStepBffrDSComm
					OR eOpsStep = MagConvLDStepMagMtyDSComm
					OR eOpsStep = MagConvLDStepBffrExitBrd
					OR eOpsStep = MagConvLDStepMagEntMESStdByChk AND (p_tyResponseFromMES.iAcceptCondition < 0 OR fbReadRFIDTO.Q))
					AND NOT(p_bOpsTravLifLDEntBrd OR p_bOpsTravLifLDUSMagWidthChk OR p_bOpsTravLifMove)
					AND (p_bDIInShutterClosedRS OR p_bLinkProjCurtainSenPrep);

	Act_OpsInfo;

	//Operation State
	bOpsInitDone		:= eOpsStep > MagConvLDStepInitMagConv;
	bStepMagExitedWait	:= eOpsStep = MagConvLDStepMagExitedWait;
	bStepMagVerification:= eOpsStep = MagConvLDStepVerifyMag;
	bStepMagMtyExit		:= eOpsStep = MagConvLDStepMagMtyExit;
	bStepMagUSCom 		:= eOpsStep = MagConvLDStepMagUSComm;
	bStepDSCom 			:= eOpsStep = MagConvLDStepBffrDSComm;
	bAGVCommRdy			:= (eOpsStep = MagConvLDStepMagUSComm OR eOpsStep = MagConvLDStepMagMtyDSComm OR eOpsStep = MagConvLDStepMagExitedWait
							OR eOpsStep = MagConvLDStepMagEnt OR eOpsStep = MagConvLDStepMagMtyExit) AND p_bAGVMagMcRunRdy;
	bRlsMagBtnUnmask	:= eOpsStep = MagConvLDStepMagEntMESStdByChk AND (p_tyResponseFromMES.iAcceptCondition < 0 OR fbReadRFIDTO.Q) OR fbWriteRFIDTO.Q;
	bExtMesStdByChk		:= eOpsStep = MagConvLDStepMagExtMESStdByChk;

END_ACTION
```

### OpsMagConvLD3.var - Change By Project
```iecst
(*2019-03-25*)
(**)
(*Action & State & Status*)
(**)
(*Alarm*)
VAR
	p_OpsMagConvLD3AlmData : UDINT;
	p_OpsMagConvLD3AlmData1 : UDINT;
END_VAR
(**)
(*Output*)
VAR
	p_OpsMagConvLD3StepTxt : UDINT;
	p_OpsMagConvLD3Paused : UDINT;
END_VAR
(**)
VAR
	p_OpsMagConvLD3BufferAct : UDINT;
	p_OpsMagConvLD3MagConv2ClpAct : UDINT;
	p_OpsMagConvLD3DSSMEMAAct : UDINT;
	p_OpsMagConvLD3AGVMagAct : UDINT;
	p_OpsMagConvLD3SafetyBarAct : UDINT;
END_VAR
(**)
VAR
	p_OpsMagConvLD3NewMagVerified : UDINT;
	p_OpsMagConvLD3MagMtyExit : UDINT;
	p_OpsMagConvLD3IncorrectMagModel : UDINT;
	p_OpsMagConvLD3MagSizeL : UDINT;
END_VAR
(**)
VAR
	p_OpsMagConvLD3InitDone : UDINT;
	p_OpsMagConvLD3MagBffrAvl : UDINT;
	p_OpsMagConvLD3NewMagAllw : UDINT;
	p_OpsMagConvLD3RlsMagAllw : UDINT;
	p_OpsMagConvLD3StepMagExitedWait : UDINT;
	p_OpsMagConvLD3StepUSCom : UDINT;
	p_OpsMagConvLD3StepSelClampCtrl : UDINT;
END_VAR
(**)
VAR
	p_OpsMagConvLD3USSOTAct : UDINT;
	p_OpsMagConvLD3DSSOTAct : UDINT;
	p_OpsMagConvLD3ExitedWait : UDINT;
	p_OpsMagConvLD3DSCom : UDINT;
	p_OpsMagConvLD3AGVCommRdy : UDINT;
	p_OpsMagConvLD3UnclmpDone : UDINT;
	p_OpsMagConvLD3MagAllwGo : UDINT;
	p_OpsMagConvLD3QueryWO : UDINT;
	p_OpsMagConvLD3ReadRFID : UDINT;
	p_OpsMagConvLD3WriteRFID : UDINT;
	p_OpsMagConvLD3ExtDelAutoRcp : UDINT;
	p_OpsMagConvLD3RlsMagUmask : UDINT;
	p_OpsMagConvLD3ExtMes : UDINT;
	p_OpsMagConvLD3HModChgDone : UDINT;
END_VAR
(**)
```

### Program Logical/Operations/OpsMagConvLD3 (IEC) - 1.00.0 - 

#### InputRef.var
```iecst
(*2019-04-16*)
(**)
(*General*)
VAR
	p_udiRstErr : REFERENCE TO UDINT;
	p_bEn : REFERENCE TO BOOL;
	p_bDis : REFERENCE TO BOOL;
	p_bRun : REFERENCE TO BOOL;
	p_bStop : REFERENCE TO BOOL;
	p_bStep : REFERENCE TO BOOL;
END_VAR
(**)
(*Configuration*)
VAR
	p_sProgNm : REFERENCE TO STRING[15];
	p_bNtSettingsLoadDone : REFERENCE TO BOOL;
END_VAR
(**)
VAR
	p_usiMagConv : REFERENCE TO USINT;
	p_bInfoEn : REFERENCE TO BOOL;
	p_bInfoMag1Mty : REFERENCE TO BOOL;
	p_bInfoMag2Mty : REFERENCE TO BOOL;
	p_bInfoMag3Mty : REFERENCE TO BOOL;
END_VAR
(**)
VAR
	pa_bMagDis : REFERENCE TO ARRAY[1..3] OF BOOL;
END_VAR
(**)
VAR
	p_bNewMag : REFERENCE TO BOOL;
	p_bRlsMag : REFERENCE TO BOOL;
	p_bUIP800Press3 : REFERENCE TO BOOL;
END_VAR
(**)
VAR
	p_bUSAllow : REFERENCE TO BOOL;
	p_tyBufferStat1 : REFERENCE TO tyBffrStat;
	p_tyBufferStat2 : REFERENCE TO tyBffrStat;
	p_tyBufferStat3 : REFERENCE TO tyBffrStat;
	p_tyBufferStat4 : REFERENCE TO tyBffrStat;
END_VAR
(**)
VAR
	p_bMagClampRS1 : REFERENCE TO BOOL;
	p_bMagClampRS2 : REFERENCE TO BOOL;
	p_bMagClampRS3 : REFERENCE TO BOOL;
	p_bMagClampRS4 : REFERENCE TO BOOL;
END_VAR
(**)
VAR
	p_bMagEntrySen1 : REFERENCE TO BOOL;
	p_bMagEntrySen2 : REFERENCE TO BOOL;
	p_bMagEntrySen3 : REFERENCE TO BOOL;
	p_bMagEntrySen4 : REFERENCE TO BOOL;
END_VAR
(**)
VAR
	p_bMagPresentSen1 : REFERENCE TO BOOL;
	p_bMagPresentSen2 : REFERENCE TO BOOL;
	p_bMagPresentSen3 : REFERENCE TO BOOL;
	p_bMagPresentSen4 : REFERENCE TO BOOL;
END_VAR
(**)
VAR
	p_bMagPresentSen : REFERENCE TO BOOL;
	p_bBufferMagPresent1 : REFERENCE TO BOOL;
	p_bBufferMagPresent2 : REFERENCE TO BOOL;
	p_bBufferMagPresent3 : REFERENCE TO BOOL;
	p_bBufferMagPresent4 : REFERENCE TO BOOL;
END_VAR
(**)
VAR
	p_dtBufferMagPresentTm1 : REFERENCE TO DATE_AND_TIME;
	p_dtBufferMagPresentTm2 : REFERENCE TO DATE_AND_TIME;
	p_dtBufferMagPresentTm3 : REFERENCE TO DATE_AND_TIME;
	p_dtBufferMagPresentTm4 : REFERENCE TO DATE_AND_TIME;
END_VAR
(**)
VAR
	p_eBufferStat : REFERENCE TO eBufferAction;
	p_eBufferStatus : REFERENCE TO eFBStatus;
END_VAR
(**)
VAR
	p_bBufferMagRemoved : REFERENCE TO BOOL;
END_VAR
(**)
VAR
	p_eMagConv2ClpStat : REFERENCE TO eMagConv2ClpAction;
	p_eMagConv2ClpStatus : REFERENCE TO eFBStatus;
	p_bMagConv2ClpHvMag : REFERENCE TO BOOL;
END_VAR
(**)
VAR
	p_eDSSMEMAStat : REFERENCE TO eSMEMAAction;
	p_eDSSMEMAStatus : REFERENCE TO eFBStatus;
	p_bDSSMEMAConvStart : REFERENCE TO BOOL;
END_VAR
(**)
VAR
	p_eAGVMagStat : REFERENCE TO eAGVMagAction;
	p_eAGVMagStatus : REFERENCE TO eFBStatus;
	p_bAGVMagMcRunRdy : REFERENCE TO BOOL;
	p_tyAGVToDTMag : REFERENCE TO tyTagAGVToDTMag;
END_VAR
(**)
VAR
	p_eSelClampCtrlStat : REFERENCE TO ePneuAction;
	p_eSelClampCtrlStatus : REFERENCE TO eFBStatus;
END_VAR
(**)
VAR
	p_bDIMagConvHeightSen : REFERENCE TO BOOL;
	p_bDIMagConvSelUnclampRS : REFERENCE TO BOOL;
	p_bDIMagConvCAB717Sen : REFERENCE TO BOOL;
	p_bDIMagConvSmallSen : REFERENCE TO BOOL;
	p_bDIMagConvLargeSen : REFERENCE TO BOOL;
	p_bDIInShutterClosedRS : REFERENCE TO BOOL;
END_VAR
(**)
VAR
	p_bOpsTravLifLDInitDone : REFERENCE TO BOOL;
END_VAR
(**)
VAR
	p_eUSSOTStat : REFERENCE TO eSOTAction;
	p_eUSSOTStatus : REFERENCE TO eFBStatus;
	p_bUSSOTTransporting : REFERENCE TO BOOL;
	p_bUSSOTConvStart : REFERENCE TO BOOL;
	p_bUSSOTConvStop : REFERENCE TO BOOL;
	p_bUSSOTUSRdy : REFERENCE TO BOOL;
	p_bUSSOTUSLargeMagRdy : REFERENCE TO BOOL;
END_VAR
(**)
VAR
	p_eDSSOTStat : REFERENCE TO eSOTAction;
	p_eDSSOTStatus : REFERENCE TO eFBStatus;
	p_bDSSOTConvStart : REFERENCE TO BOOL;
	p_bDSSOTConvStop : REFERENCE TO BOOL;
END_VAR
(**)
VAR
	p_bDISOTRcv : REFERENCE TO BOOL;
	p_bDISOTAGVReady : REFERENCE TO BOOL;
	p_bInShutterExtended : REFERENCE TO BOOL;
END_VAR
(**)
VAR
	p_bLD1ExitedWait : REFERENCE TO BOOL;
	p_bLD2ExitedWait : REFERENCE TO BOOL;
	p_bLD4ExitedWait : REFERENCE TO BOOL;
END_VAR
(**)
VAR
	p_eSafetyBarStat : REFERENCE TO ePneuAction;
	p_eSafetyBarStatus : REFERENCE TO eFBStatus;
	p_bSafetyBarExtended : REFERENCE TO BOOL;
	p_bSafetyBarRetracted : REFERENCE TO BOOL;
	p_bOpsTravLifULUpdatePullSlot : REFERENCE TO BOOL;
	p_eOpsTravLifLDPosGo : REFERENCE TO eTravLifLDPos;
	p_bOpsTravLifErrCmdUnclmp : REFERENCE TO BOOL;
	p_bProjLifTravMnlLoad : REFERENCE TO BOOL;
	p_bOpsTravLifLDEntBrd : REFERENCE TO BOOL;
	p_bOpsTravLifLDUSMagWidthChk : REFERENCE TO BOOL;
	p_bOpsTravLifMove : REFERENCE TO BOOL;
	p_bEjectMag : REFERENCE TO BOOL;
END_VAR
(**)
(**)
```

#### InputRef_Link.var
```iecst
(*2020-05-20*)
(**)
(*External Data*)
VAR
	p_bLinkDIMagPresentSen1 : REFERENCE TO BOOL;
	p_bLinkMagConv2Clp1MtrIn : REFERENCE TO BOOL;
	p_bLinkMagConv2Clp1MtrOut : REFERENCE TO BOOL;
	p_bLinkDIMagPresentSen2 : REFERENCE TO BOOL;
	p_bLinkMagConv2Clp2MtrIn : REFERENCE TO BOOL;
	p_bLinkMagConv2Clp2MtrOut : REFERENCE TO BOOL;
	p_bLinkDIMagPresentSen3 : REFERENCE TO BOOL;
	p_bLinkMagConv2Clp3MtrIn : REFERENCE TO BOOL;
	p_bLinkMagConv2Clp3MtrOut : REFERENCE TO BOOL;
	p_bLinkDIMagPresentSen4 : REFERENCE TO BOOL;
	p_bLinkMagConv2Clp4MtrIn : REFERENCE TO BOOL;
	p_bLinkMagConv2Clp4MtrOut : REFERENCE TO BOOL;
	p_bLinkFixedMagClampRS1 : REFERENCE TO BOOL;
	p_bLinkRmtMagClampRS1 : REFERENCE TO BOOL;
	p_bLinkFixedMagClampRS2 : REFERENCE TO BOOL;
	p_bLinkRmtMagClampRS2 : REFERENCE TO BOOL;
	p_bLinkFixedMagClampRS3 : REFERENCE TO BOOL;
	p_bLinkRmtMagClampRS3 : REFERENCE TO BOOL;
	p_bLinkFixedMagClampRS4 : REFERENCE TO BOOL;
	p_bLinkRmtMagClampRS4 : REFERENCE TO BOOL;
	p_bLinkMcParamMagAutoDetTm : REFERENCE TO DINT;
	p_bLinkDIMagEntrySen : REFERENCE TO BOOL;
	p_bLinkNtParamMagModelAutoVerify : REFERENCE TO BOOL;
	p_bLinkMagRcpCurrRcpMagModel : REFERENCE TO USINT;
	p_bLinkNewMagVerified1 : REFERENCE TO BOOL;
	p_bLinkNewMagVerified2 : REFERENCE TO BOOL;
	p_bLinkNewMagVerified4 : REFERENCE TO BOOL;
END_VAR
(**)
VAR
	p_eLinkMag : REFERENCE TO eLDMag;
	p_usiLinkMod : REFERENCE TO USINT;
	p_bLinkMagRcpCurrRcpMagModel1 : REFERENCE TO USINT;
	p_bLinkProjCurtainSenPrep : REFERENCE TO BOOL;
	p_eLinkMcParamMagExMode : REFERENCE TO eMcMagExchangeMode;
	p_bMag3OrientationChkSen1 : REFERENCE TO BOOL;
	p_bMagOrientChkSenPrep : REFERENCE TO BOOL;
	p_bMagHeightDetSen3 : REFERENCE TO BOOL;
	p_bMagHeightDetEn : REFERENCE TO BOOL;
	p_bMagHeightDetPrep : REFERENCE TO BOOL;
	p_bFixedSideDetect : REFERENCE TO BOOL;
END_VAR
(**)
VAR
	p_eNtParamCustomerReq : REFERENCE TO eCustomer;
	p_bHermesSvyPrep : REFERENCE TO BOOL;
	p_bMcParamHermesSvyEn : REFERENCE TO BOOL;
	p_bMcParamMesRFIDEn : REFERENCE TO BOOL;
	p_diRFIDTO : REFERENCE TO DINT;
	p_bMagPropDiffBlk : REFERENCE TO BOOL;
	p_bNtParamAutoRcpPrep : REFERENCE TO BOOL;
	p_bAutoRcpbMag3RcpLoaded : REFERENCE TO BOOL;
	p_ausiSvyMagAccOrder : REFERENCE TO ARRAY[1..3] OF USINT;
END_VAR
(*Siemen MES*)
VAR
	p_tyResponseFromMES : REFERENCE TO tyStatPlatformFromMES;
	p_bHCommModChg : REFERENCE TO BOOL;
END_VAR
(*We_Fabricate*)
VAR
	p_ausiLCSLFMagAccOrder : REFERENCE TO ARRAY[1..3] OF USINT;
END_VAR
```

#### Local.var
```iecst
(*2019-04-16*)
(**)
(*Local Action, State & Status*)
VAR
	eStatus : eFBStatus := Idle;
	udiStatus : UDINT := 0;
	udiStatus1 : UDINT := 0;
END_VAR
(**)
(*Local Alarm*)
VAR
	tyAlmData : tyAlmDat;
	tyAlmData1 : tyAlmDat;
	a_tyAlmText : ARRAY[10000..10099] OF tyAlmTxt := [(sAlmText:='Magazine Not Present'),(sAlmText:='Magazine 1 Is Empty'),(sAlmText:='Magazine 2 Is Empty'),(sAlmText:='Magazine 3 Is Empty'),(sAlmText:='Wrong Magazine Width On Position 3'),(sAlmText:='Wrong Magazine Height On Position 3'),(sAlmText:='Waiting for Unload Magazine 3'),(0),(sAlmText:='Wrong Magazine Orientation Placed Or Wrong Magazine Loaded',sRcyText:='Please Check And Correct the Magazine Orientation/Reload Correct Magazine.'),(sAlmText:='MES response to Write RFID Timeout, Press Release Mag to Manual Exit'),4((0)),(sAlmText:='Writing Mag 3 RFID'),(sAlmText:='Writing Mag 3 RFID or Press Release Mag'),(sAlmText:='Wrong Magazine Position 3.Press Release Magazine To Continue.'),83((0))];
END_VAR
(**)
(*Local Output*)
VAR
	sStepTxt : STRING[80];
	bPaused : BOOL;
END_VAR
(**)
VAR
	eBufferAct : eBufferAction;
	eSelClampCtrl : ePneuAction;
	eMagConv2ClpAct : eMagConv2ClpAction;
	eDSSMEMAAct : eSMEMAAction;
	eAGVMagAct : eAGVMagAction;
	eSafetyBarAct : ePneuAction;
	eUSSOTAct : eSOTAction;
	eDSSOTAct : eSOTAction;
	bOpsInitDone : BOOL;
	bMagBffrAvl : BOOL;
	bNewMagAllw : BOOL;
	bRlsMagAllw : BOOL;
	bStepMagExitedWait : BOOL;
	bStepMagVerification : BOOL;
	bStepMagMtyExit : BOOL;
	bStepMagUSCom : BOOL;
	bStepMagCmp : BOOL;
	bPneuUnclmpDone : BOOL;
	bQueryWO : BOOL;
END_VAR
VAR RETAIN
	usiAccWO : INT;
	iMagMESAcptCond : INT;
END_VAR
(*ForSiemen*)
VAR
	ePrevStepBeforeMESStdBy : eMagConvLDStep := MagConvLDStepNA;
END_VAR
VAR RETAIN
	bWriteRFID : BOOL;
END_VAR
VAR
	bReadRFID : BOOL;
	fbReadRFIDTO : TON := (PT:=T#3s);
	fbWriteRFIDTO : TON := (PT:=T#5s);
END_VAR
(**)
(*Local Input*)
VAR
	udiRstErr : UDINT := 0;
	bEn : BOOL := TRUE;
	bDis : BOOL := FALSE;
	bRun : BOOL;
	bStop : BOOL;
	bStep : BOOL;
	usiMagConv : USINT;
	bInfoEn : BOOL;
	bInfoMag1Mty : BOOL;
	bInfoMag2Mty : BOOL;
	bInfoMag3Mty : BOOL;
	a_bMagDis : ARRAY[1..4] OF BOOL;
	bNewMag : BOOL;
	bRlsMag : BOOL;
	bUSAllow : BOOL;
	tyBufferStat1 : tyBffrStat;
	tyBufferStat2 : tyBffrStat;
	tyBufferStat3 : tyBffrStat;
	tyBufferStat4 : tyBffrStat;
	bMagClampRS1 : BOOL;
	bMagClampRS2 : BOOL;
	bMagClampRS3 : BOOL;
	bMagClampRS4 : BOOL;
	bMagEntrySen1 : BOOL;
	bMagEntrySen2 : BOOL;
	bMagEntrySen3 : BOOL;
	bMagEntrySen4 : BOOL;
	bMagPresentSen1 : BOOL;
	bMagPresentSen2 : BOOL;
	bMagPresentSen3 : BOOL;
	bMagPresentSen4 : BOOL;
	bBufferMagPresent1 : BOOL;
	bBufferMagPresent2 : BOOL;
	bBufferMagPresent3 : BOOL;
	bBufferMagPresent4 : BOOL;
	dtBufferMagPresentTm1 : DATE_AND_TIME;
	dtBufferMagPresentTm2 : DATE_AND_TIME;
	dtBufferMagPresentTm3 : DATE_AND_TIME;
	dtBufferMagPresentTm4 : DATE_AND_TIME;
	eBufferStat : eBufferAction;
	eBufferStatus : eFBStatus;
	eMagConv2ClpStat : eMagConv2ClpAction;
	eMagConv2ClpStatus : eFBStatus;
	bMagConv2ClpHvMag : BOOL;
	eDSSMEMAStat : eSMEMAAction;
	eDSSMEMAStatus : eFBStatus;
	bDSSMEMAConvStart : BOOL;
	eAGVMagStat : eAGVMagAction;
	eAGVMagStatus : eFBStatus;
	bAGVMagMcRunRdy : BOOL;
	tyAGVToDTMag : tyTagAGVToDTMag;
	diRFIDTO : DINT := 5000;
	sProgNm : STRING[15] := 'Ops MagConvUL';
	bNtSettingsLoadDone : BOOL := TRUE;
END_VAR
(**)
(*Local*)
VAR
	bRstErr : BOOL;
	udiRstErrOld : UDINT;
	bInitDone : BOOL;
	bInitialDone : BOOL;
	eOpsStep : eMagConvLDStep := MagConvLDStepNA;
	eGotoOpsStep : eMagConvLDStep := MagSetupULStepInitPneu;
	bMagMtyExitedWait : BOOL;
	udi : UDINT;
	udi1 : UDINT;
	udiCount : UDINT;
	udiCmpTm : UDINT;
	udiMagAllwGo : UDINT;
	a_tyMagAllwBffrStat : ARRAY[1..4] OF tyBffrStat;
	a_bMagAllwMagClamped : ARRAY[1..4] OF BOOL;
	a_bMagAllwMagPresent : ARRAY[1..4] OF BOOL;
	a_udiMagAllwMagPresentTm : ARRAY[1..4] OF UDINT;
	a_udiMagAllwPriority : ARRAY[1..4] OF UDINT;
	a_udiMagAllwSum : ARRAY[1..4] OF UDINT;
	p_tyLocalBufferStat : REFERENCE TO tyBffrStat;
	p_bLocalMagEntrySen : REFERENCE TO BOOL;
	p_bLocalBufferMagPresent : REFERENCE TO BOOL;
	p_dtLocalBufferMagPresentTm : REFERENCE TO DATE_AND_TIME;
END_VAR
(**)
VAR
	fbWrongMagTm : TON := (PT:=T#5000ms);
	fbSelClmpTm : TON := (PT:=T#1s); (*No Ret sensor*)
	fbMagAutoDetTm : TON := (PT:=T#2000ms);
	fbMagRemovedTm : TON := (PT:=T#2000ms);
	fbEntSenOff : TON := (PT:=T#1000ms);
	fbVerifyWarningDelay : TON := (PT:=T#1000ms);
	bNewMagAutoDetected : BOOL;
	bNewMagVerified : BOOL;
	bNewMagVerifyStarted : BOOL;
	bIncorrectMagazineModel : BOOL;
	bSetMagFull : BOOL;
	bMagToAGVAvailable : BOOL;
	bWrongHeight : BOOL;
	bWrongWidth : BOOL;
	bMagSizeLarge : BOOL;
	bLimitSenActivated : BOOL;
END_VAR
VAR RETAIN
	bManualUnloadMag : BOOL;
END_VAR
VAR
	bAIVInPos : BOOL;
END_VAR
VAR RETAIN
	bMagExitedWait : BOOL;
END_VAR
VAR
	usiMagModel : USINT;
	bMagManEx : BOOL;
	bMagAutoEx : BOOL;
	bStepDSCom : BOOL;
	bOpsTravLifULUpdatePullSlot : BOOL;
	bAGVCommRdy : BOOL;
	bExitDelAutoRcp : BOOL;
	bRlsMagBtnUnmask : BOOL;
	bExtMesStdByChk : BOOL;
	bHCommModChgDone : BOOL;
END_VAR
(*Step Logger*)
VAR
	bClsLog : BOOL;
	blog : BOOL;
	logStep : ARRAY[0..999] OF eMagConvLDStep;
	logIndexStep : INT;
	eGotoOpsStepDummy : eMagConvLDStep;
	udiModuleNum : UDINT := 6071;
END_VAR
(**)
(**)
```

#### Act_InitGlobal.st
```iecst
(** 2019-04-16 **)
ACTION Act_InitGlobal:

	(* Always Change If Project Change *)

	//Pass Data To Link
	p_bLinkDIMagPresentSen1 ACCESS p_DIMagPresentSen1;
	p_bLinkMagConv2Clp1MtrIn ACCESS p_MagConv2Clp1MtrSigOnOrLToR;
	p_bLinkMagConv2Clp1MtrOut ACCESS p_MagConv2Clp1MtrDirOrRToL;
	p_bLinkDIMagPresentSen2 ACCESS p_DIMagPresentSen2;
	p_bLinkMagConv2Clp2MtrIn ACCESS p_MagConv2Clp2MtrSigOnOrLToR;
	p_bLinkMagConv2Clp2MtrOut ACCESS p_MagConv2Clp2MtrDirOrRToL;
	p_bLinkDIMagPresentSen3 ACCESS p_DIMagPresentSen3;
	p_bLinkMagConv2Clp3MtrIn ACCESS p_MagConv2Clp3MtrSigOnOrLToR;
	p_bLinkMagConv2Clp3MtrOut ACCESS p_MagConv2Clp3MtrDirOrRToL;
	p_bLinkDIMagPresentSen3 ACCESS p_DIMagPresentSen3;
	p_bLinkMagConv2Clp3MtrIn ACCESS p_MagConv2Clp3MtrSigOnOrLToR;
	p_bLinkMagConv2Clp3MtrOut ACCESS p_MagConv2Clp3MtrDirOrRToL;
	p_bLinkDIMagPresentSen4 ACCESS p_DIMagPresentSen4;
	p_bLinkMagConv2Clp4MtrIn ACCESS p_MagConv2Clp4MtrSigOnOrLToR;
	p_bLinkMagConv2Clp4MtrOut ACCESS p_MagConv2Clp4MtrDirOrRToL;

	p_bLinkFixedMagClampRS1 ACCESS p_DIMag1FixedClampRS;
	p_bLinkRmtMagClampRS1 ACCESS p_DIMag1RemoteClampRS;

	p_bLinkFixedMagClampRS2 ACCESS p_DIMag2FixedClampRS;
	p_bLinkRmtMagClampRS2 ACCESS p_DIMag2RemoteClampRS;

	p_bLinkFixedMagClampRS3 ACCESS p_DIMag3FixedClampRS;
	p_bLinkRmtMagClampRS3 ACCESS p_DIMag3RemoteClampRS;

	p_bLinkFixedMagClampRS4 ACCESS p_DIMag4FixedClampRS;
	p_bLinkRmtMagClampRS4 ACCESS p_DIMag4RemoteClampRS;

	p_bLinkDIMagEntrySen ACCESS p_DIMagConvEntSen3;
	p_bLinkMcParamMagAutoDetTm ACCESS p_McParamMagAutoDetTm;
	p_bLinkNtParamMagModelAutoVerify ACCESS p_NtParamProjMagAutoVerifyPrep;
	p_bLinkMagRcpCurrRcpMagModel ACCESS p_MagRcpCurrRcpMagModel;

	p_bLinkNewMagVerified1 ACCESS p_OpsMagConvLD1NewMagVerified;
	p_bLinkNewMagVerified2 ACCESS p_OpsMagConvLD2NewMagVerified;
	p_bLinkNewMagVerified4 ACCESS p_OpsMagConvLD4NewMagVerified;

	p_eLinkMag ACCESS p_NtParamProjMag;
	p_usiLinkMod ACCESS p_ProdRcpCurrRcp1McMod;
	p_bLinkMagRcpCurrRcpMagModel1 ACCESS p_MagRcpCurrRcpMagModel1;

	p_bLinkProjCurtainSenPrep ACCESS p_NtParamProjCurtainSenPrep;
	p_eLinkMcParamMagExMode ACCESS p_McParamMagExMode;
	p_bMag3OrientationChkSen1 ACCESS p_DIMag3OrientChkSen1;
	p_bMagOrientChkSenPrep ACCESS p_NtParamProjMagOrientChkSenPrep;
	p_bMagHeightDetSen3 ACCESS p_DIHighMagDetSen3;
	p_bMagHeightDetEn ACCESS p_MagRcpCurrRcpMagHeightChkEn;
	p_bMagHeightDetPrep	ACCESS p_NtParamProjMagHeightChkPrep;
	p_bFixedSideDetect ACCESS p_DIMag3FixedSideDetect;//sensor

	p_eNtParamCustomerReq ACCESS p_NtParamCustomerReq;
	p_bHermesSvyPrep ACCESS p_NtParamHermesSvyPrep; //queryWO
	p_bNtParamAutoRcpPrep ACCESS p_NtParamAutoRcpPrep;
	p_bMcParamHermesSvyEn ACCESS p_McParamHermesSvyEn;
	p_bMcParamMesRFIDEn ACCESS p_McParamMesRFIDEn;		//MES Rfid opcua
	p_diRFIDTO ACCESS p_McParamMesRFIDTOInMS;

	p_bMagPropDiffBlk ACCESS p_AutoRcpbMag3PropDiffBlk; //link- false
	p_bAutoRcpbMag3RcpLoaded ACCESS p_AutoRcpbMag3RcpLoaded; //ops
	p_ausiSvyMagAccOrder ACCESS p_SvyHermesMagAccOrder;
	p_tyResponseFromMES ACCESS p_TagFromMesMagConv3; //For Siemen
	p_bHCommModChg ACCESS p_UIHCommModChg;

	p_ausiLCSLFMagAccOrder ACCESS p_LCSLFMagAccOrder;

	//Pass Data To Internal Use
	p_udiRstErr ACCESS p_RstErrReset;
	p_bEn ACCESS p_NtParamProjMag3ConvPrep;
	p_bRun ACCESS p_OpsRun;
	p_bStop ACCESS p_OpsStop;
	p_bStep ACCESS p_OpsStep;

	p_sProgNm ACCESS p_NtParamOpsMagConvLD3ProgNm;
	p_bNtSettingsLoadDone ACCESS p_StartupNtSettingsLoadDone;

	pa_bMagDis ACCESS p_OpsTravLifLDMagDis;

	p_bNewMag ACCESS p_UINewMag3;
	p_bRlsMag ACCESS p_UIRlsMag3;
	p_bUIP800Press3 ACCESS p_UIP800Press3;

	p_tyBufferStat1 ACCESS p_Buffer1BffrStat;
	p_tyBufferStat2 ACCESS p_Buffer2BffrStat;
	p_tyBufferStat3 ACCESS p_Buffer3BffrStat;
	p_tyBufferStat4 ACCESS p_Buffer4BffrStat;

	p_bMagEntrySen1 ACCESS p_DIMagConvEntSen1;
	p_bMagEntrySen2 ACCESS p_DIMagConvEntSen2;
	p_bMagEntrySen3 ACCESS p_DIMagConvEntSen3;
	p_bMagEntrySen4 ACCESS p_DIMagConvEntSen4;

	p_bMagPresentSen ACCESS p_Buffer3MagPresent;
	p_bBufferMagPresent1 ACCESS p_Buffer1MagPresent;
	p_bBufferMagPresent2 ACCESS p_Buffer2MagPresent;
	p_bBufferMagPresent3 ACCESS p_Buffer3MagPresent;
	p_bBufferMagPresent4 ACCESS p_Buffer4MagPresent;

	p_dtBufferMagPresentTm1 ACCESS p_Buffer1MagPresentTm;
	p_dtBufferMagPresentTm2 ACCESS p_Buffer2MagPresentTm;
	p_dtBufferMagPresentTm3 ACCESS p_Buffer3MagPresentTm;
	p_dtBufferMagPresentTm4 ACCESS p_Buffer4MagPresentTm;

	p_eBufferStat ACCESS p_Buffer3Stat;
	p_eBufferStatus ACCESS p_Buffer3Status;

	p_bBufferMagRemoved ACCESS p_Buffer3MagRemoved;

	p_eMagConv2ClpStat ACCESS p_MagConv2Clp3Stat;
	p_eMagConv2ClpStatus ACCESS p_MagConv2Clp3Status;
	p_bMagConv2ClpHvMag ACCESS p_MagConv2Clp3HvMag;

	p_eDSSMEMAStat ACCESS p_DSSMEMA3Stat;
	p_eDSSMEMAStatus ACCESS p_DSSMEMA3Status;
	p_bDSSMEMAConvStart ACCESS p_DSSMEMA3ConvStart;

	p_eAGVMagStat ACCESS p_AGVMag3Stat;
	p_eAGVMagStatus ACCESS p_AGVMag3Status;
	p_bAGVMagMcRunRdy ACCESS p_AGVMag3McRunRdy;
	p_tyAGVToDTMag ACCESS p_AGVTagAGVToDTMag;

	p_eSelClampCtrlStat ACCESS p_PneuNoSenSelClamp3Stat;
	p_eSelClampCtrlStatus ACCESS p_PneuNoSenSelClamp3Status;

	p_bDIMagConvHeightSen ACCESS p_DIMagConvHeightSen3;
	p_bDIMagConvSelUnclampRS ACCESS p_DIMag3SelUnclampRS;
	p_bDIMagConvCAB717Sen ACCESS p_DIMagConvCAB717MagSen3;
	p_bDIMagConvSmallSen ACCESS p_DIMagConvSmallMagSen3;
	p_bDIMagConvLargeSen ACCESS p_DIMagConvLargeMagSen3;
	p_bDIInShutterClosedRS ACCESS p_DIInShutterCloseRS;

	p_bOpsTravLifLDInitDone ACCESS p_OpsTravLifLDInitDone;

	//USSOT
	p_eUSSOTStat ACCESS p_USSOT3Stat;
	p_eUSSOTStatus ACCESS p_USSOT3Status;
	p_bUSSOTTransporting ACCESS p_USSOT3Transporting;
	p_bUSSOTConvStart ACCESS p_USSOT3ConvStart;
	p_bUSSOTConvStop ACCESS p_USSOT3ConvStop;
	p_bUSSOTUSRdy ACCESS p_USSOT3USRdy;
	p_bUSSOTUSLargeMagRdy ACCESS p_USSOT3USLargeMagRdy;

	//DSSOT
	p_eDSSOTStat ACCESS p_DSSOT3Stat;
	p_eDSSOTStatus ACCESS p_DSSOT3Status;
	p_bDSSOTConvStart ACCESS p_DSSOT3ConvStart;
	p_bDSSOTConvStop ACCESS p_DSSOT3ConvStop;

	p_bDISOTRcv ACCESS p_DISOT3Receive;
	p_bDISOTAGVReady ACCESS p_DISOT3Ready;

	p_bInShutterExtended ACCESS p_Pneu2SenInShutterExtended3;

	p_bUSAllow ACCESS p_Follower1USAllow;

	p_bLD1ExitedWait ACCESS p_OpsMagConvLD1ExitedWait;
	p_bLD2ExitedWait ACCESS p_OpsMagConvLD2ExitedWait;
	p_bLD4ExitedWait ACCESS p_OpsMagConvLD4ExitedWait;

	p_eSafetyBarStat ACCESS p_Pneu2SMag3SafetyBarStat;
	p_eSafetyBarStatus ACCESS p_Pneu2SMag3SafetyBarStatus;
	p_bSafetyBarExtended ACCESS p_Pneu2SMag3SafetyBarExtended;
	p_bSafetyBarRetracted ACCESS p_Pneu2SMag3SafetyBarRetracted;

	p_bOpsTravLifULUpdatePullSlot ACCESS p_OpsTravLifULUpdatePullSlot;
	p_eOpsTravLifLDPosGo ACCESS p_OpsTravLifLDPosGo;

	p_bOpsTravLifErrCmdUnclmp ACCESS p_OpsTravLifWChkErrCmdUnclmp3;
	p_bProjLifTravMnlLoad	ACCESS p_NtParamProjLifTravMnlLoad;

	p_bOpsTravLifLDEntBrd ACCESS p_OpsTravLifLDEntBrd;
	p_bOpsTravLifLDUSMagWidthChk ACCESS p_OpsTravLifLDUSMagWidthChk;
	p_bOpsTravLifMove ACCESS p_OpsTravLifMove;

	p_bEjectMag ACCESS p_UIEjectMag3;

	(* Always Change If Project Change *)

END_ACTION
```

#### Act_Initial.st
```iecst
(** 2019-01-20 **)
ACTION Act_Initial:

	//Initial
	IF p_bLinkDIMagPresentSen3 THEN
		bSetMagFull := TRUE;
	END_IF

END_ACTION
```

#### Act_InitLocal.st
```iecst
(** 2019-04-16 **)
ACTION Act_InitLocal:

	//Input Reference Link To Local Variable
	p_udiRstErr ACCESS ADR(udiRstErr);
	p_bEn ACCESS ADR(bEn);
	p_bDis ACCESS ADR(bDis);
	p_bRun ACCESS ADR(bRun);
	p_bStop ACCESS ADR(bStop);
	p_bStep ACCESS ADR(bStep);

	p_sProgNm ACCESS ADR(sProgNm);
	p_bNtSettingsLoadDone ACCESS ADR(bNtSettingsLoadDone);

	p_usiMagConv ACCESS ADR(usiMagConv);
	p_bInfoEn ACCESS ADR(bInfoEn);
	p_bInfoMag1Mty ACCESS ADR(bInfoMag1Mty);
	p_bInfoMag2Mty ACCESS ADR(bInfoMag2Mty);
	p_bInfoMag3Mty ACCESS ADR(bInfoMag3Mty);

	pa_bMagDis ACCESS ADR(a_bMagDis);

	p_bNewMag ACCESS ADR(bNewMag);
	p_bRlsMag ACCESS ADR(bRlsMag);

	p_bUSAllow ACCESS ADR(bUSAllow);
	p_tyBufferStat1 ACCESS ADR(tyBufferStat1);
	p_tyBufferStat2 ACCESS ADR(tyBufferStat2);
	p_tyBufferStat3 ACCESS ADR(tyBufferStat3);
	p_tyBufferStat4 ACCESS ADR(tyBufferStat4);

	p_bMagClampRS1 ACCESS ADR(bMagClampRS1);
	p_bMagClampRS2 ACCESS ADR(bMagClampRS2);
	p_bMagClampRS3 ACCESS ADR(bMagClampRS3);
	p_bMagClampRS4 ACCESS ADR(bMagClampRS4);

	p_bMagEntrySen1 ACCESS ADR(bMagEntrySen1);
	p_bMagEntrySen2 ACCESS ADR(bMagEntrySen2);
	p_bMagEntrySen3 ACCESS ADR(bMagEntrySen3);
	p_bMagEntrySen4 ACCESS ADR(bMagEntrySen4);

	p_bMagPresentSen1 ACCESS ADR(bMagPresentSen1);
	p_bMagPresentSen2 ACCESS ADR(bMagPresentSen2);
	p_bMagPresentSen3 ACCESS ADR(bMagPresentSen3);
	p_bMagPresentSen4 ACCESS ADR(bMagPresentSen4);

	p_bBufferMagPresent1 ACCESS ADR(bBufferMagPresent1);
	p_bBufferMagPresent2 ACCESS ADR(bBufferMagPresent2);
	p_bBufferMagPresent3 ACCESS ADR(bBufferMagPresent3);
	p_bBufferMagPresent4 ACCESS ADR(bBufferMagPresent4);

	p_dtBufferMagPresentTm1 ACCESS ADR(dtBufferMagPresentTm1);
	p_dtBufferMagPresentTm2 ACCESS ADR(dtBufferMagPresentTm2);
	p_dtBufferMagPresentTm3 ACCESS ADR(dtBufferMagPresentTm3);
	p_dtBufferMagPresentTm4 ACCESS ADR(dtBufferMagPresentTm4);

	p_eBufferStat ACCESS ADR(eBufferStat);
	p_eBufferStatus ACCESS ADR(eBufferStatus);

	p_eMagConv2ClpStat ACCESS ADR(eMagConv2ClpStat);
	p_eMagConv2ClpStatus ACCESS ADR(eMagConv2ClpStatus);
	p_bMagConv2ClpHvMag ACCESS ADR(bMagConv2ClpHvMag);

	p_eDSSMEMAStat ACCESS ADR(eDSSMEMAStat);
	p_eDSSMEMAStatus ACCESS ADR(eDSSMEMAStatus);
	p_bDSSMEMAConvStart ACCESS ADR(bDSSMEMAConvStart);

	p_eAGVMagStat ACCESS ADR(eAGVMagStat);
	p_eAGVMagStatus ACCESS ADR(eAGVMagStatus);
	p_bAGVMagMcRunRdy ACCESS ADR(bAGVMagMcRunRdy);
	p_tyAGVToDTMag ACCESS ADR(tyAGVToDTMag);

	p_diRFIDTO ACCESS ADR(diRFIDTO);

END_ACTION
```

#### Act_Link.st
```iecst
(** 2018-12-11 **)
ACTION Act_Link:

	IF p_eLinkMag = LDMagQuadruple = FALSE THEN
		//Sensor
		p_bMagPresentSen1	:= p_bLinkDIMagPresentSen1 OR p_bLinkMagConv2Clp1MtrIn OR p_bLinkMagConv2Clp1MtrOut;
		p_bMagPresentSen2	:= p_bLinkDIMagPresentSen2 OR p_bLinkMagConv2Clp2MtrIn OR p_bLinkMagConv2Clp2MtrOut;
		p_bMagPresentSen3	:= p_bLinkDIMagPresentSen3 OR p_bLinkMagConv2Clp3MtrIn OR p_bLinkMagConv2Clp3MtrOut;
		p_bMagPresentSen4	:= p_bLinkDIMagPresentSen4 OR p_bLinkMagConv2Clp4MtrIn OR p_bLinkMagConv2Clp4MtrOut;
		//Clamp RS
		p_bMagClampRS1 		:= (p_bLinkFixedMagClampRS1 AND p_bLinkRmtMagClampRS1) OR p_bLinkNewMagVerified1;
		p_bMagClampRS2		:= (p_bLinkFixedMagClampRS2 AND p_bLinkRmtMagClampRS2) OR p_bLinkNewMagVerified2;
		p_bMagClampRS3		:= (p_bLinkFixedMagClampRS3 AND p_bLinkRmtMagClampRS3) OR bNewMagVerified;
		p_bMagClampRS4		:= (p_bLinkFixedMagClampRS4 AND p_bLinkRmtMagClampRS4) OR p_bLinkNewMagVerified4;
	ELSE
		IF p_eLinkMag = LDMagQuadruple THEN
			CASE p_usiLinkMod OF
				0,1:
					//Sensor
					p_bMagPresentSen1	:= p_bLinkDIMagPresentSen1 OR p_bLinkMagConv2Clp1MtrIn OR p_bLinkMagConv2Clp1MtrOut;
					p_bMagPresentSen2	:= p_bLinkDIMagPresentSen2 OR p_bLinkMagConv2Clp2MtrIn OR p_bLinkMagConv2Clp2MtrOut;
					p_bMagPresentSen3	:= p_bLinkDIMagPresentSen3 OR p_bLinkMagConv2Clp3MtrIn OR p_bLinkMagConv2Clp3MtrOut;
					p_bMagPresentSen4	:= p_bLinkDIMagPresentSen4 OR p_bLinkMagConv2Clp4MtrIn OR p_bLinkMagConv2Clp4MtrOut;
					//Clamp RS
					p_bMagClampRS1 		:= (p_bLinkFixedMagClampRS1 AND p_bLinkRmtMagClampRS1) OR p_bLinkNewMagVerified1;
					p_bMagClampRS2		:= (p_bLinkFixedMagClampRS2 AND p_bLinkRmtMagClampRS2) OR p_bLinkNewMagVerified2;
					p_bMagClampRS3		:= (p_bLinkFixedMagClampRS3 AND p_bLinkRmtMagClampRS3) OR bNewMagVerified;
					p_bMagClampRS4		:= (p_bLinkFixedMagClampRS4 AND p_bLinkRmtMagClampRS4) OR p_bLinkNewMagVerified4;

				2:

					//Sensor
					p_bMagPresentSen1	:= FALSE;
					p_bMagPresentSen2	:= FALSE;
					p_bMagPresentSen3	:= p_bLinkDIMagPresentSen3 OR p_bLinkMagConv2Clp3MtrIn OR p_bLinkMagConv2Clp3MtrOut;
					p_bMagPresentSen4	:= p_bLinkDIMagPresentSen4 OR p_bLinkMagConv2Clp4MtrIn OR p_bLinkMagConv2Clp4MtrOut;
					//Clamp RS
					p_bMagClampRS1 		:= FALSE;
					p_bMagClampRS2		:= FALSE;
					p_bMagClampRS3		:= (p_bLinkFixedMagClampRS3 AND p_bLinkRmtMagClampRS3) OR bNewMagVerified;
					p_bMagClampRS4		:= (p_bLinkFixedMagClampRS4 AND p_bLinkRmtMagClampRS4) OR p_bLinkNewMagVerified4;

			END_CASE
		END_IF
	END_IF

	//Mag Exchange Mode
	CASE p_eLinkMcParamMagExMode OF
		McSetMagXcAutoManMode:
			bMagManEx := TRUE;
			bMagAutoEx := TRUE;

		McSetMagXcAutoMode:
			bMagManEx := FALSE;
			bMagAutoEx := TRUE;

		McSetMagXcManMode:
			bMagManEx := TRUE;
			bMagAutoEx := FALSE;

	END_CASE

	//New magazine auto detection at inlet sensor
	fbMagAutoDetTm(IN := p_bLinkDIMagEntrySen  OR p_bLinkDIMagPresentSen3, PT := DINT_TO_TIME(p_bLinkMcParamMagAutoDetTm));
	IF fbMagAutoDetTm.Q AND bMagManEx THEN
		bNewMagAutoDetected := TRUE;
	ELSE
		bNewMagAutoDetected := FALSE;
	END_IF

	//Front or rear lane magazine mode
	IF p_eLinkMag = LDMagQuadruple THEN
		CASE p_usiLinkMod OF
			0:
				usiMagModel := p_bLinkMagRcpCurrRcpMagModel;

			1,2:
				usiMagModel := p_bLinkMagRcpCurrRcpMagModel1;
		END_CASE

	ELSE
		usiMagModel := p_bLinkMagRcpCurrRcpMagModel;

	END_IF

	IF p_bLinkNtParamMagModelAutoVerify THEN
		IF usiMagModel = 0  //CAB706.2
			AND p_bDIMagConvHeightSen = TRUE
			AND p_bDIMagConvSelUnclampRS = FALSE
			AND p_bDIMagConvCAB717Sen = FALSE
			AND p_bDIMagConvSmallSen
			THEN
			bNewMagVerified:= TRUE;

		ELSIF  usiMagModel = 1 //CAB716.2
			AND p_bDIMagConvHeightSen = FALSE
			AND p_bDIMagConvSelUnclampRS = FALSE
			AND p_bDIMagConvCAB717Sen = FALSE
			AND p_bDIMagConvSmallSen
			THEN
			bNewMagVerified:= TRUE;

		ELSIF  usiMagModel = 2 //CAB717.2
			AND p_bDIMagConvHeightSen = FALSE
			AND p_bDIMagConvSelUnclampRS
			AND p_bDIMagConvCAB717Sen
			AND p_bDIMagConvLargeSen
			THEN
			bNewMagVerified:= TRUE;
		ELSE
			bNewMagVerified:= FALSE;
		END_IF
	ELSE
		bNewMagVerified:= TRUE;
	END_IF

	bAIVInPos := p_tyAGVToDTMag.bVEHInPos3 OR p_bDISOTRcv;

	IF p_bBufferMagRemoved THEN
		bManualUnloadMag := FALSE;
	END_IF

	IF EDGEPOS(p_bOpsTravLifULUpdatePullSlot) THEN
		bOpsTravLifULUpdatePullSlot := TRUE;
	ELSIF p_bOpsTravLifULUpdatePullSlot = FALSE THEN
		bOpsTravLifULUpdatePullSlot := FALSE;
	END_IF

	//Auto recipe
	IF p_bNtParamAutoRcpPrep THEN
		p_bUSAllow := NOT(p_bMagPropDiffBlk); //false
//		p_bAdaptFollowerBlk := p_sProdRcpCurrRcp1Name <>  p_sProdRcpCrZ2RcpNm;
	ELSE
		p_bUSAllow ACCESS p_Follower1USAllow;
//		p_bAdaptFollowerBlk := FALSE;
	END_IF

END_ACTION
```

#### Init.st
```iecst
(** 2019-03-25 **)
PROGRAM _INIT

	(* Always Change If Project Change *)

	//Physical Configuration
	usiMagConv	:= 3;

	//Pass Address To Global Address For External Use
	//Action, State & Status

	//Alarm
	p_OpsMagConvLD3AlmData	:= ADR(tyAlmData);
	p_OpsMagConvLD3AlmData1	:= ADR(tyAlmData1);

	//Output
	p_OpsMagConvLD3StepTxt				:= ADR(sStepTxt);
	p_OpsMagConvLD3Paused				:= ADR(bPaused);

	p_OpsMagConvLD3BufferAct			:= ADR(eBufferAct);
	p_OpsMagConvLD3MagConv2ClpAct		:= ADR(eMagConv2ClpAct);
	p_OpsMagConvLD3DSSMEMAAct			:= ADR(eDSSMEMAAct);
	p_OpsMagConvLD3AGVMagAct			:= ADR(eAGVMagAct);
	p_OpsMagConvLD3SafetyBarAct			:= ADR(eSafetyBarAct);

	p_OpsMagConvLD3InitDone				:= ADR(bOpsInitDone);
	p_OpsMagConvLD3MagBffrAvl			:= ADR(bMagBffrAvl);
	p_OpsMagConvLD3NewMagAllw			:= ADR(bNewMagAllw);
	p_OpsMagConvLD3RlsMagAllw			:= ADR(bRlsMagAllw);
	p_OpsMagConvLD3StepMagExitedWait	:= ADR(bStepMagExitedWait);
	p_OpsMagConvLD3StepUSCom			:= ADR(bStepMagUSCom);

	p_OpsMagConvLD3StepSelClampCtrl		:= ADR(eSelClampCtrl);

	p_OpsMagConvLD3NewMagVerified		:= ADR(bNewMagVerified);
	p_OpsMagConvLD3MagMtyExit			:= ADR(bStepMagMtyExit);
	p_OpsMagConvLD3IncorrectMagModel    := ADR(bIncorrectMagazineModel);
	p_OpsMagConvLD3MagSizeL    			:= ADR(bMagSizeLarge);

	p_OpsMagConvLD3USSOTAct			:= ADR(eUSSOTAct);
	p_OpsMagConvLD3DSSOTAct			:= ADR(eDSSOTAct);

	p_OpsMagConvLD3ExitedWait			:= ADR(bMagExitedWait);
	p_OpsMagConvLD3DSCom				:= ADR(bStepDSCom);
	p_OpsMagConvLD3AGVCommRdy			:= ADR(bAGVCommRdy);

	p_OpsMagConvLD3UnclmpDone			:= ADR(bPneuUnclmpDone);
	p_OpsMagConvLD3MagAllwGo			:= ADR(udiMagAllwGo);
	p_OpsMagConvLD3QueryWO 				:= ADR(bQueryWO);
	p_OpsMagConvLD3ReadRFID				:= ADR(bReadRFID);
	p_OpsMagConvLD3WriteRFID			:= ADR(bWriteRFID);
	p_OpsMagConvLD3ExtDelAutoRcp		:= ADR(bExitDelAutoRcp);
	p_OpsMagConvLD3RlsMagUmask			:= ADR(bRlsMagBtnUnmask);
	p_OpsMagConvLD3ExtMes				:= ADR(bExtMesStdByChk);
	p_OpsMagConvLD3HModChgDone			:= ADR(bHCommModChgDone);

	(* Always Change If Project Change *)

END_PROGRAM
```

#### Program Logical/Operations/OpsMagConvLD3/Sequence

##### Act_OpsInfo.st
```iecst
ACTION Act_OpsInfo:

	//Reset
	udiStatus1	:= 0;

	//Magazine Verification Warning
	fbMagRemovedTm(IN:= p_bMagPresentSen = FALSE AND p_bLocalMagEntrySen = FALSE AND p_bBufferMagRemoved);
	IF fbMagRemovedTm.Q OR bNewMagVerified THEN
		bNewMagVerifyStarted := FALSE;
	END_IF

	fbVerifyWarningDelay(IN:= bNewMagVerifyStarted AND bNewMagVerified = FALSE AND bStepMagVerification = FALSE);

	IF fbVerifyWarningDelay.Q AND p_tyBufferStat3.bBffrMty = FALSE THEN
		IF bManualUnloadMag = FALSE THEN
			CASE usiMagModel OF
				0: //CAB706.2
					IF bWrongHeight THEN
						udiStatus1	:= 10005;
					ELSIF p_bDIMagConvHeightSen = FALSE THEN
						bWrongHeight := TRUE;

					ELSIF bWrongWidth THEN
						udiStatus1	:= 10004;
					ELSIF p_bDIMagConvSelUnclampRS
						OR p_bDIMagConvCAB717Sen
						OR p_bDIMagConvSmallSen = FALSE
						THEN
						bWrongWidth := TRUE;
					END_IF

				1: //CAB716.2
					IF bWrongHeight THEN
						udiStatus1	:= 10005;
					ELSIF p_bDIMagConvHeightSen = TRUE THEN
						bWrongHeight := TRUE;

					ELSIF bWrongWidth THEN
						udiStatus1	:= 10004;
					ELSIF p_bDIMagConvSelUnclampRS
						OR p_bDIMagConvCAB717Sen
						OR p_bDIMagConvSmallSen = FALSE
						THEN
						bWrongWidth := TRUE;
					END_IF

				2: //CAB717.2
					IF bWrongHeight THEN
						udiStatus1	:= 10005;
					ELSIF p_bDIMagConvHeightSen THEN
						bWrongHeight := TRUE;

					ELSIF bWrongWidth THEN
						udiStatus1	:= 10004;
					ELSIF p_bDIMagConvSelUnclampRS = FALSE
						OR p_bDIMagConvCAB717Sen = FALSE
						OR p_bDIMagConvLargeSen
						THEN
						bWrongWidth := TRUE;

					END_IF

			END_CASE
		ELSIF bManualUnloadMag THEN
			udiStatus1	:= 10006;
		END_IF

	ELSIF 	udiStatus1 <> 10004
		AND udiStatus1 <> 10005
		AND p_tyBufferStat3.bBffrMty = FALSE
		AND bStepMagExitedWait
		AND p_bLocalMagEntrySen
		THEN
		udiStatus1	:= 10006;
		bManualUnloadMag := TRUE;
	ELSE
		bWrongHeight := FALSE;
		bWrongWidth	:= FALSE;
	END_IF

	bIncorrectMagazineModel := udiStatus1 = 10004 OR udiStatus1 = 10005;

	//----------------------------Siemens MES -------------------------------------//
	IF (udiStatus1 = 0) AND p_eNtParamCustomerReq = Siemens OR p_eNtParamCustomerReq = We_Fabricate THEN
		IF eOpsStep = MagConvLDStepMagExtMESStdByChk   THEN //we_fab no use
			IF NOT(fbWriteRFIDTO.Q) THEN
				udiStatus1 := 10014;
			ELSIF fbWriteRFIDTO.Q THEN
				udiStatus1 := 10015;
			END_IF
			IF (fbMagRemovedTm.Q ) THEN
				fbWriteRFIDTO(IN:= FALSE);
			END_IF
		ELSIF eOpsStep = MagConvLDStepMagEntMESStdByChk THEN
			IF p_tyResponseFromMES.iAcceptCondition < 0 THEN
				udiStatus1 := 10016; //wrong magazine position x.Press Release Magazine To Continue.
			END_IF
		END_IF

	END_IF

END_ACTION
```

##### Act_OpsRst.st
```iecst
(** 2019-03-25 **)
ACTION Act_OpsRst:

	udiStatus1	:= 0;

	eBufferAct		:= BufferActIdle;
	eMagConv2ClpAct	:= MagConv2ClpActIdle;
	eDSSMEMAAct		:= SMEMAActIdle;
	eAGVMagAct		:= AGVMagActIdle;
	eSelClampCtrl	:= PneuActIdle;
	eDSSOTAct		:= SOTActIdle;
	eUSSOTAct		:= SOTActIdle;
	eSafetyBarAct	:= PneuActIdle;

	bNewMagVerified := FALSE;
	bNewMagVerifyStarted := FALSE;

END_ACTION
```
